	(*TERMINAL 50KF1 (EL6001 Interface (RS232))  ********1-Channel Serial Interface RS232***********************)
	ib50A1_EL6001PortNo								AT %I* :  UINT;
	ist50A1_HandScannerCOMPortDataIn				AT %I* :  EL6InData22B;
	qst50A1_HandScannerCOMPortDataOut				AT %Q*: EL6OutData22B;

	(*TERMINAL 60KF1 (EL1008 8Ch. Dig. Input 24V, 3ms) ******************************************************)
	ib60KF1_1_Spare 								AT %I*: BOOL;
	ib60KF1_5_Spare									AT %I*: BOOL;
	ib60KF1_2_Spare									AT %I*: BOOL;
	ib60KF1_6_Spare									AT %I*: BOOL;
	ib60KF1_3_Spare 								AT %I*: BOOL;
	ib60KF1_7_Spare									AT %I*: BOOL;
	ib60KF1_4_Spare									AT %I*: BOOL;
	ib60KF1_8_Spare 	 							AT %I*: BOOL;

	(*TERMINAL 61KF1 (EL1008 8Ch. Dig. Input 24V, 3ms) ******************************************************)
	ib61KF1_1_DoorOpenZone1_SFCP					AT %I*: BOOL;
	ib61KF1_5_DoorOpenZone2_SFCP					AT %I*: BOOL;
	ib61KF1_2_CasePackerAutoRun_SFCP  				AT %I*: BOOL;
	ib61KF1_6_CaseRejected_SFCP		 				AT %I*: BOOL;
	ib61KF1_3_RowComplete_SFCP  					AT %I*: BOOL;
	ib61KF1_7_LayerComplete_SFCP  					AT %I*: BOOL;
	ib61KF1_4_CaseComplete_SFCP  					AT %I*: BOOL;
	ib61KF1_8_CaseDischarged_SFCP  					AT %I*: BOOL;

	(*TERMINAL 62KF1 (EL1008 8Ch. Dig. Input 24V, 3ms) ******************************************************)
	ib62KF1_1_CasePresentPosition01_SFCP								AT %I*: BOOL;
	ib62KF1_5_CasePresentPosition02_SFCP								AT %I*: BOOL;
	ib62KF1_2_CasePresentPosition03_SFCP						AT %I*: BOOL;
	ib62KF1_6_CasePresentPosition04_SFCP							AT %I*: BOOL;
	ib62KF1_3_CasePresentPosition05_SFCP							AT %I*: BOOL;
	ib62KF1_7_CasePresentPosition06_SFCP							AT %I*: BOOL;
	ib62KF1_4_CasePresentPosition07_SFCP								AT %I*: BOOL;
	ib62KF1_8_CasePresentPosition08_SFCP							AT %I*: BOOL;

	(*TERMINAL 63KF1 (EL1008 8Ch. Dig. Input 24V, 3ms) ******************************************************)
	ib63KF1_1_24VPowerSupplyOK 						AT %I*: BOOL;
	ib63KF1_5_EthernetSwitchOK 						AT %I*: BOOL;	 (* Option *)
	ib63KF1_2_CaseLabelValidationTrig_SFCP 			AT %I*: BOOL;
	ib63KF1_6_QAButtonRejectOuter_SFCP 				AT %I*: BOOL;
	ib63KF1_3_IntermediatePush_SFCP 				AT %I*: BOOL;
	ib63KF1_7_24VPowerSupplyAdditionalUnitOK			AT %I*: BOOL;
	ib63KF1_4_CasePresentPrintAreaSensor			AT %I*: BOOL;	 (* Option *)
	ib63KF1_8_CaseLeavingPrintAreaSensor			AT %I*: BOOL;	 (* Option *)

	(*TERMINAL 64KF1 (EL1008 8Ch. Dig. Input 24V, 3ms) ******************************************************)
	ib64KF1_1_PackSeparationDriveOK					AT %I*: BOOL;
	ib64KF1_5_Spare							AT %I*: BOOL;	(*  *)
	ib64KF1_2_IntermediateCameraTrigSesnorOK						AT %I*: BOOL;	(*  *)
	ib64KF1_6_AdditionalConveyorPlugConnected					AT %I*: BOOL;	(*  *)
	ib64KF1_3_OutfeedConveyorPlugConnected			AT %I*: BOOL; (**)
	ib64KF1_7_TransferConveyorPlugConnected			AT %I*: BOOL;	(* *)
	ib64KF1_4_Guard1 								AT %I*: BOOL; 	(* *)
	ib64KF1_8_Guard2								AT %I*: BOOL; 	(**)

	(*TERMINAL 65KF1 (EL1008 8Ch. Dig. Input 24V, 3ms) ******************************************************)
	ib65KF1_1_PSRisReset							AT %I*: BOOL;
	ib65KF1_5_PSRisOK								AT %I*: BOOL;
	ib65KF1_2_EmergencyStopFromPSR					AT %I*: BOOL;
	ib65KF1_6_EmergencyCircuitFromPSR 				AT %I*: BOOL;
	ib65KF1_3_AirDumpStatus					AT %I*: BOOL; 	(*  *)
	ib65KF1_7_Guard3								AT %I*: BOOL; 	(*  *)
	ib65KF1_4_Guard4								AT %I*: BOOL; 	(*   *)
	ib65KF1_8_Guard5								AT %I*: BOOL; 	(*  *)

	(*TERMINAL 66KF1 (EL1008 8Ch. Dig. Input 24V, 3ms) ******************************************************)
	ib66KF1_1_AirSupplyOK									AT %I*: BOOL;
	ib66KF1_5_PreMachineInAutorun					AT %I*: BOOL;		(*coneccted - input in PreMachine plug 18DX1 *)
	ib66KF1_2_PostMachineInAutorun					AT %I*: BOOL;		(*not coneccted - input in Safety plug 18DX2 *)
	ib66KF1_6_OuterRejectConfirmation				AT %I*: BOOL;		(*Duplicated*)
	ib66KF1_3_MainConveyorStart						AT %I*: BOOL;
	ib66KF1_7_CaseRejctConfirmCameraInReadCycle	AT %I*: BOOL;
	ib66KF1_4_CaseRejctConfirmCameraNoRead		AT %I*: BOOL;
	ib66KF1_8_CaseRejctConfirmCameraGoodRead		AT %I*: BOOL;

	(*TERMINAL 67KF1 (EL1008 8Ch. Dig. Input 24V, 3ms) ******************************************************)
	ib67KF1_1_Spare									AT %I*: BOOL;
	ib67KF1_5_Spare									AT %I*: BOOL;
	ib67KF1_2_Spare									AT %I*: BOOL;
	ib67KF1_6_Spare									AT %I*: BOOL;
	ib67KF1_3_Spare									AT %I*: BOOL;
	ib67KF1_7_Spare									AT %I*: BOOL;
	ib67KF1_4_Spare									AT %I*: BOOL;
	ib67KF1_8_Spare									AT %I*: BOOL;

	(*TERMINAL 69KF1 (EL1008 8Ch. Dig. Input 24V, 3ms) ******************************************************)
	ib69KF1_1_Labeller01Ready							AT %I*: BOOL;
	ib69KF1_5_Labeller01DataReady						AT %I*: BOOL;
	ib69KF1_2_Labeller01HomePosition							AT %I*: BOOL;
	ib69KF1_6_Labeller01LabelPrinted							AT %I*: BOOL;
	ib69KF1_3_Labeller01SummaryWarning							AT %I*: BOOL;
	ib69KF1_7_Labeller01Error								AT %I*: BOOL;
	ib69KF1_4_Labeller01AirPressureOK							AT %I*: BOOL;
	ib69KF1_8_Labeller01InPosition						AT %I*: BOOL;

	(*TERMINAL 70KF1 (EL1008 8Ch. Dig. Input 24V, 3ms) ******************************************************)
	ib70KF1_1_MainsSupplyHealthy					AT %I*: BOOL;	(*  *)
	ib70KF1_5_UPSHealthy							AT %I*: BOOL;	(*  *)
	ib70KF1_2_UPSBatteryMode						AT %I*: BOOL;	(*  *)
	ib70KF1_6_UPSBatteryCharging					AT %I*: BOOL;	(*  *)
	ib70KF1_3_Spare									AT %I*: BOOL; (**)
	ib70KF1_7_Spare								AT %I*: BOOL;	(* *)
	ib70KF1_4_Spare 								AT %I*: BOOL; 	(* *)
	ib70KF1_8_Spare								AT %I*: BOOL; 	(* *)

	(*TERMINAL 80KF1 (EL2008 8Ch. Dig. Output 24V, 0.5A) ******************************************************)
	qb80KF1_1_LightPoleGREEN  						AT %Q*: BOOL;
	qb80KF1_5_LightPoleAMBER  						AT %Q*: BOOL;
	qb80KF1_2_LightPoleRED  						AT %Q*: BOOL;
	qb80KF1_6_LightPoleALARM  						AT %Q*: BOOL;	 (* Option *)
	qb80KF1_3_LightHandscannerBoxGreen 				AT %Q*: BOOL;	 (* Option *)
	qb80KF1_7_LightHandscannerBoxRed  				AT %Q*: BOOL;	 (* Option *)
	qb80KF1_4_Spare  								AT %Q*: BOOL;
	qb80KF1_8_OuterRejectSignal   					AT %Q*: BOOL;	 (*Option*)

	(*TERMINAL 81KF1 (EL2008 8Ch. Dig. Output 24V, 0.5A) ******************************************************)
	qb81KF1_1_SafetyReset	  						AT %Q*: BOOL;
	qb81KF1_5_PackSeperationDriveFaultAck			AT %Q*: BOOL;
	qb81KF1_2_PackSeperationDriveBrakeRelease		AT %Q*: BOOL;	 (* Option *)
	qb81KF1_6_CaseRejctConfirmCameraPower 								AT %Q*: BOOL;
	qb81KF1_3_CaseRejctConfirmCameraTrigger									AT %Q*: BOOL;
	qb81KF1_7_PreMachineAddditionalCutOut			AT %Q*: BOOL;	 (* not coneccted - output in Safety plug 18DX1  *)
	qb81KF1_4_PreMachineCutOut						AT %Q*: BOOL;	(*coneccted - output in PreMachine plug 18DX1 *)
	qb81KF1_8_PostMachineAddditionalCutOut	 					AT %Q*: BOOL;		(* not coneccted - output in PostMachine Safety plug 18DX2 *)

	(*TERMINAL 82KF1 (EL2008 8Ch. Dig. Output 24V, 0.5A) ******************************************************)
	qb82KF1_1_PostMachineCutOut_STCP		  					AT %Q*: BOOL;		(*coneccted - output in PostMachine plug 19DX2 *)
	qb82KF1_5_CaseValidationOK_STCP					AT %Q*: BOOL;
	qb82KF1_2_OuterValidationOK_STCP 				AT %Q*: BOOL;
	qb82KF1_6_CaseContentOK_STCP					AT %Q*: BOOL;
	qb82KF1_3_LabellerInhibit_STL					AT %Q*: BOOL;
	qb82KF1_7_RejectSignal3_STL 					AT %Q*: BOOL;	(*  *)
	qb82KF1_4_Miscellaneous_STL						AT %Q*: BOOL;	(*  *)
	qb82KF1_8_Spare			 						AT %Q*: BOOL;

	(*TERMINAL 83KF1 (EL2008 8Ch. Dig. Output 24V, 0.5A) ******************************************************)
	qb83KF1_1_PackSepparationDriveRun									AT %Q*: BOOL;
	qb83KF1_5_AdditionalConveyor01Run									AT %Q*: BOOL;
	qb83KF1_2_AdditionalConveyor02Run									AT %Q*: BOOL;
	qb83KF1_6_Spare									AT %Q*: BOOL;
	qb83KF1_3_Spare									AT %Q*: BOOL;
	qb83KF1_7_Spare									AT %Q*: BOOL;
	qb83KF1_4_Spare									AT %Q*: BOOL;
	qb83KF1_8_Labeller01DoorGuardOpen			AT %Q*: BOOL;

	(*TERMINAL 84KF1 (EL2008 8Ch. Dig. Output 24V, 0.5A) ******************************************************)
	qb84KF1_1_Spare								AT %Q*: BOOL;
	qb84KF1_5_Spare									AT %Q*: BOOL;
	qb84KF1_2_Spare									AT %Q*: BOOL;
	qb84KF1_6_Spare									AT %Q*: BOOL;
	qb84KF1_3_Spare									AT %Q*: BOOL;
	qb84KF1_7_Spare									AT %Q*: BOOL;
	qb84KF1_4_Spare									AT %Q*: BOOL;
	qb84KF1_8_Spare									AT %Q*: BOOL;

	(*TERMINAL 88KF1 (EL4002 2Ch. Analog Output, 0…10 V, 12 bit) ******************************************************)
	qn88KF1_1_PackSeparationDriveCh1							AT %Q* : INT;
	qn88KF1_2_Spare											AT %Q* : INT;

	(*TERMINAL 90KF1 (EL2624 4Ch. Relay Output, 125 V AC, 30 V DC, 0.5 A AC, 2 A DC)******************)
	qb90KF1_1_Labeller01ResetSignal					AT %Q*: BOOL;		(**)
	qb90KF1_2_Labeller01PrintSignal							AT %Q*: BOOL;		(**)
	qb90KF1_3_Labeller01ApplySignal1						AT %Q*: BOOL;		(**)
	qb90KF1_4_Labeller01ApplySignal2										AT %Q*: BOOL;

	(*TERMINAL 97KF1 - EL6631 -  PROFINET IO Controller ********************************************************)
	ist97KF1_Master01PNetState 						AT %I* : ST_CX_EtherCATMasterPNetState;

	(*DRIVE  3T1  - G120C ************************************************************************************)
	ist3T1_outerseparation							AT %I* : ST_DRIVE_INPUT;
	qst3T1_outerseparation							AT %Q* : ST_DRIVE_OUTPUT;

	(*DRIVE  4T1  - G120C ************************************************************************************)
	ist4T1_transferconveyor							AT %I* : ST_DRIVE_INPUT;
	qst4T1_transferconveyor							AT %Q* : ST_DRIVE_OUTPUT;

	(*DRIVE  5T1  - G120C ************************************************************************************)
	ist5T1_outfeedconveyor							AT %I* : ST_DRIVE_INPUT;
	qst5T1_outfeedconveyor							AT %Q* : ST_DRIVE_OUTPUT;

	(*DRIVE  6T1  - G120C ************************************************************************************)
	ist6T1_additionalconveyor						AT %I* : ST_DRIVE_INPUT;
	qst6T1_additionalconveyor					AT %Q* : ST_DRIVE_OUTPUT;
END_VAR

// ---- Global Variables/InputsOutputs_OC/IOVariablesEUCA_OC.TcGVL
{attribute 'Tc2GvlVarNames'}
VAR_GLOBAL

(*TERMINAL XXXKF1 - EK1100 **********************************************************)

(*TERMINAL 350KF1 (EL6001 Interface (RS232))  ********1-Channel Serial Interface RS232***********************)
	ib350A1_EL6001PortNo								AT %I* :  UINT;
	ist350A1_HandScannerCOMPortDataIn					AT %I* :  EL6InData22B;
	qst350A1_HandScannerCOMPortDataOut					AT %Q*: EL6OutData22B;

(*TERMINAL 351KF1 - EL4002 ******************************************************)
	qn351KF1_1_OuterValidationLightingIntensity			AT %Q* : INT;
	qn351KF1_2_OuterAggregationLightingIntensity		AT %Q* : INT;

(*TERMINAL 352KF1 - EL4002 ******************************************************)
	qn352KF1_1_CaseContentValidationLightingIntensity	AT %Q* : INT;
	qn352KF1_2_LightingIntensity							AT %Q* : INT;

(*TERMINAL 360KF1 - EL1008 ***********************************************************)
	ib360KF1_1_OuterAtInfeed							AT %I* : BOOL;	(* Option *)
	ib360KF1_5_OuterInfeedBlocked						AT %I* : BOOL;	(* Option clamp*)
	ib360KF1_2_OuterAtLabeller							AT %I* : BOOL;	(* Option gate*)
	ib360KF1_6_PackConfirmationCameraTrigSensor			AT %I* : BOOL;
	ib360KF1_3_OuterValidationCameraTrigSensor 					AT %I* : BOOL;
	ib360KF1_7_OuterAtReject							AT %I* : BOOL;
	ib360KF1_4_RejectConfirmation						AT %I* : BOOL;
	ib360KF1_8_RejectBinFull								AT %I* : BOOL;

(*TERMINAL 361KF1 - EL1008 ***********************************************************)
	ib361KF1_1_OuterClampExtended							AT %I* : BOOL;
	ib361KF1_5_OuterGateExtended					AT %I* : BOOL;
	ib361KF1_2_OuterGateRetracted						AT %I* : BOOL;
	ib361KF1_6_OuterGateImpactSensor						AT %I* : BOOL;
	ib361KF1_3_RejectCylinderExtended					AT %I* : BOOL;
	ib361KF1_7_RejectCylinderRetracted					AT %I* : BOOL;
	ib361KF1_4_EUCAExitBlocked										AT %I* : BOOL;	(* Option *)
	ib361KF1_8_EUCABuildBack									AT %I* : BOOL;

(*TERMINAL 362KF1 - EL1008 ************************************************************)
	ib362KF1_1_Labeller02Ready							AT %I*: BOOL;
	ib362KF1_5_Labeller02DataReady						AT %I*: BOOL;
	ib362KF1_2_Labeller02HomePosition 			AT %I*: BOOL;
	ib362KF1_6_Labeller02LabelPrinted						AT %I*: BOOL;
	ib362KF1_3_Labeller02SummaryWarning					AT %I*: BOOL;
	ib362KF1_7_Labeller02Error							AT %I*: BOOL;
	ib362KF1_4_Labeller02AirPressureOK							AT %I*: BOOL;
	ib362KF1_8_Labeller02InPosition					AT %I*: BOOL;	(* ??? *)

(*TERMINAL 363KF1 (EL1008 8Ch. Dig. Input 24V, 3ms) ***************************************)
	ib363KF1_1_QAButtonRejectOuter						AT %I*: BOOL;	(* Option *)
	ib363KF1_5_IntermediatePushSensor					AT %I*: BOOL;
	ib363KF1_2_CaseLabelValidationCameraTrigSensor 		AT %I*: BOOL;
	ib363KF1_6_OuterAggregationCameraTrigSensor			AT %I*: BOOL;	(* *)
	ib363KF1_3_RowCompleteSensor						AT %I*: BOOL;
	ib363KF1_7_LayerCompleteSensor						AT %I*: BOOL;
	ib363KF1_4_CaseCompleteSensor						AT %I*: BOOL;
	ib363KF1_8_CaseDischargedSensor						AT %I*: BOOL;

(*TERMINAL 366KF1 (EL1008 8Ch. Dig. Input 24V, 3ms) ****************************************)
	ib366KF1_1_OuterAtAdditionalConveyor02									AT %I*: BOOL;
	ib366KF1_5_ExitBlockedAdditionalConveyor02									AT %I*: BOOL;
	ib366KF1_2_Spare									AT %I*: BOOL;
	ib366KF1_6_Spare									AT %I*: BOOL;
	ib366KF1_3_Spare									AT %I*: BOOL;
	ib366KF1_7_Spare									AT %I*: BOOL;
	ib366KF1_4_Spare								AT %I*: BOOL;
	ib366KF1_8_RemoteAirSupplyOK									AT %I*: BOOL;

(*TERMINAL 380KF1 - EL2008 (EL2008 8Ch. Dig. Output 24V, 0.5A) ********************************)
	qb380KF1_1_ClampCylinderExtend				AT %Q*: BOOL;
	qb380KF1_5_Spare						 			AT %Q*: BOOL;
	qb380KF1_2_GateCylinderExtend 						AT %Q*: BOOL;		(**)
	qb380KF1_6_GateCylinderRetract	 					AT %Q*: BOOL;		(**)
	qb380KF1_3_RejectCylinderExtend						AT %Q*: BOOL;
	qb380KF1_7_RejectCylinderRetract			  		AT %Q*: BOOL;
	qb380KF1_4_Spare								AT %Q*: BOOL;
	qb380KF1_8_PLCControlledAggCameraLightning			AT %Q*: BOOL; (**)

(*TERMINAL 381KF1 (EL2008 8Ch. Dig. Output 24V, 0.5A) ***************************************)
	qb381KF1_1_RearConfirmationCameraTrigger			AT %Q*: BOOL;
	qb381KF1_5_RearConfirmationCameraPower				AT %Q*: BOOL;
	qb381KF1_2_FrontConfirmationCameraTrigger			AT %Q*: BOOL;
	qb381KF1_6_FrontConfirmationCameraPower	 			AT %Q*: BOOL;
	qb381KF1_3_OuterValidationCameraTrig 					AT %Q*: BOOL;
	qb381KF1_7_OuterValidationCameraPower				AT %Q*: BOOL;
	qb381KF1_4_OuterAggregationCameraTrig					AT %Q*: BOOL;
	qb381KF1_8_OuterAggregationCameraPower					AT %Q*: BOOL;

(*TERMINAL 382KF1 (EL2008 8Ch. Dig. Output 24V, 0.5A) ****************************************)
	qb382KF1_1_CaseContentValidationCameraTrig				AT %Q*: BOOL;
	qb382KF1_5_CaseContentValidationCameraPower			AT %Q*: BOOL;
	qb382KF1_2_CaseLabelValidationCameraTrig				AT %Q*: BOOL;
	qb382KF1_6_CaseLabelValidationCameraPower	 			AT %Q*: BOOL;
	qb382KF1_3_OuterValidationCameraLightning					AT %Q*: BOOL;		(**)
	qb382KF1_7_OuterAggregationCameraLightning				AT %Q*: BOOL;		(**)
	qb382KF1_4_CaseContentValidationCameraLightning			AT %Q*: BOOL;		(**)
	qb382KF1_8_Labeller02DoorGuardOpen				AT %Q*: BOOL;		(**)

(*TERMINAL 390KF1 (EL2624 4Ch. Relay Output, 125 V AC, 30 V DC, 0.5 A AC, 2 A DC)******************)
	qb390KF1_1_Labeller02ResetSignal						AT %Q*: BOOL;
	qb390KF1_2_Labeller02PrintSignal						AT %Q*: BOOL;
	qb390KF1_3_Labeller02ApplySignal1						AT %Q*: BOOL;
	qb390KF1_4_Labeller02ApplySignal2								AT %Q*: BOOL;

END_VAR

// ---- Global Variables/InputsOutputs_OC/IOVariablesPAOL_OC.TcGVL
{attribute 'Tc2GvlVarNames'}
VAR_GLOBAL

(*TERMINAL XXXKF1 - EK1100 ******************************************************)

(*TERMINAL 647KF1 - EL4002 ******************************************************)
	qn647KF1_1_LightingIntensity							AT %Q* : INT;
	qn647KF1_2_Spare									AT %Q* : INT;

(*TERMINAL 660KF1 - EL1008 ******************************************************)
	ib660KF1_1_PackAggregationCameraRigTrigger			AT %I* : BOOL;
	ib660KF1_5_PackAggregationCamera1Trigger				AT %I* : BOOL;
	ib660KF1_2_PackAggregationCamera2Trigger				AT %I* : BOOL;
	ib660KF1_6_PackAggregationCamera3Trigger				AT %I* : BOOL;
	ib660KF1_3_PreMachineBuildBack						AT %I* : BOOL;
	ib660KF1_7_TPDExitBlock								AT %I* : BOOL;
	ib660KF1_4_PackAggregationCamera4Trigger				AT %I* : BOOL;	(* Option *)
	ib660KF1_8_PackIsolatorDrive							AT %I* : BOOL;

(*TERMINAL 680KF1 - EL2008 ******************************************************)
	qb680KF1_1_PackAggregationCamera1Enable				AT %Q* : BOOL;
	qb680KF1_5_PackAggregationCamera2Enable				AT %Q* : BOOL;
	qb680KF1_2_PackAggregationCamera3Enable				AT %Q* : BOOL;
	qb680KF1_6_PackAggregationCamera1Power				AT %Q* : BOOL;
	qb680KF1_3_PackAggregationCamera2Power				AT %Q* : BOOL;
	qb680KF1_7_PackAggregationCamera3Power				AT %Q* : BOOL;
	qb680KF1_4_PackAggregationCamera4Enable				AT %Q* : BOOL;
	qb680KF1_8_PackCamerasLenseAir						AT %Q* : BOOL;

END_VAR

// ---- Global Variables/InputsOutputs_OC/IOVariablesPLAS_OC.TcGVL
{attribute 'Tc2GvlVarNames'}
VAR_GLOBAL

(*TERMINAL XXXKF1 - EK1100 ******************************************************)


(*TERMINAL 747KF1 - EL4002 ******************************************************)
	qn747KF1_1_LightingIntensityPackAggregationCamera							AT %Q* : INT;
	qn747KF1_2_LightingIntensityPackConfirmationCamera							AT %Q* : INT;

(*TERMINAL 748KF1 - EL4002 ******************************************************)
	qn748KF1_1_LightingIntensityMasterListCamera		AT %Q* : INT;
	qn748KF1_2_Spare										AT %Q* : INT;

(*TERMINAL 763KF1 - EL1008 ******************************************************)
	ib763KF1_1_MasterListCameraTrigSensor					AT %I* : BOOL;
	ib763KF1_5_SpareMasterListCameraTrigSensor			AT %I* : BOOL;		(* Option *)
	ib763KF1_2_AggregationCameraTrigSensor				AT %I* : BOOL;
	ib763KF1_6_SpareAggregationCamera1TrigSensor		AT %I* : BOOL;		(* Option *)
	ib763KF1_3_SpareAggregationCamera2TrigSensor		AT %I* : BOOL;		(* Option *)
	ib763KF1_7_PackQueueIndex								AT %I* : BOOL; 		(* Option *)
	ib763KF1_4_StackQueueIndex								AT %I* : BOOL; 		(* Option *)
	ib763KF1_8_SpareIndex											AT %I* : BOOL;

(*TERMINAL 764KF1 - EL1008 ******************************************************)
	ib764KF1_1_OuterIndexComplete							AT %I* : BOOL;
	ib764KF1_5_SpareCameraTrigSesnor						AT %I* : BOOL;		(* Option *)
	ib764KF1_2_Guard1 										AT %I* : BOOL;		(*FOCKE/GD Master list guard*)
	ib764KF1_6_Guard2										AT %I* : BOOL;		(*FOCKE/GD Master list guard*)
	ib764KF1_3_Guard3 										AT %I* : BOOL;		(*FOCKE/GD Aggregation guard*)
	ib764KF1_7_Guard4 										AT %I* : BOOL;		(*FOCKE/GD Aggregationt guard*)
	ib764KF1_4_OuterBrushOpen								AT %I* : BOOL;
	ib764KF1_8_RejectTowerActive							AT %I* : BOOL;

(*TERMINAL 765KF1 (EL1008 8Ch. Dig. Input 24V, 3ms) ******************************************************)
	ib765KF1_1_FilmInPosition 								AT %I*: BOOL;
	ib765KF1_5_SparePrinterTrigger							AT %I*: BOOL;
	ib765KF1_2_IntermediateCamera1TrigSesnor				AT %I*: BOOL;
	ib765KF1_6_HeatTunelPackReject							AT %I*: BOOL;
	ib765KF1_3_OuterAtAdditionalConveyor01 				AT %I*: BOOL;
	ib765KF1_7_IntermediateCamera2TrigSesnor				AT %I*: BOOL;
	ib765KF1_4_OuterAtReject									AT %I*: BOOL;		(*AdditionalConveyor01*)
	ib765KF1_8_RejectConfirmation	 						AT %I*: BOOL;		(*AdditionalConveyor01*)

(*TERMINAL 766KF1 - EL1008 ******************************************************)
	ib766KF1_1_RejectCylinderExtended						AT %I* : BOOL;
	ib766KF1_5_RejectCylinderRetracted						AT %I* : BOOL;		(*  *)
	ib766KF1_2_RejectBinFull 									AT %I* : BOOL;		(*AdditionalConveyor01*)
	ib766KF1_6_ExitBlockedAdditionalConveyor01				AT %I* : BOOL;
	ib766KF1_3_IntermediateCamera3TrigSesnor				AT %I* : BOOL;
	ib766KF1_7_Spare											AT %I* : BOOL;	(*Potentially for GD Additional Master list guard*)
	ib766KF1_4_Spare											AT %I* : BOOL;		(* Guard5 Potentially for GD Wrapper door*)
	ib766KF1_8_Spare											AT %I* : BOOL;			(* Guard6 Potentially for GD Wrapper door*)

(*TERMINAL 767KF1 - EL1008 ******************************************************)
	ib767KF1_1_ConveyorInterfaceInputSignal1				AT %I* : BOOL;
	ib767KF1_5_ConveyorInterfaceInputSignal2				AT %I* : BOOL;		(*  *)
	ib767KF1_2_RejectTower2Active							AT %I* : BOOL;		(**)
	ib767KF1_6_Spare											AT %I* : BOOL;
	ib767KF1_3_Spare											AT %I* : BOOL;
	ib767KF1_7_Spare 											AT %I* : BOOL;
	ib767KF1_4_Spare											AT %I* : BOOL;
	ib767KF1_8_Spare											AT %I* : BOOL;


(*TERMINAL 783KF1 - EL2008 ******************************************************)
	qb783KF1_1_MasterListCameraPower						AT %Q* : BOOL;
	qb783KF1_5_SpareMasterListCameraPower					AT %Q* : BOOL;	(* Option *)
	qb783KF1_2_SpareAggregationCameraPower				AT %Q* : BOOL;	(* Option *)
	qb783KF1_6_AggregationCamera1Power					AT %Q* : BOOL;
	qb783KF1_3_AggregationCamera2Power					AT %Q* : BOOL;
	qb783KF1_7_ConfirmationCamera1Power					AT %Q* : BOOL; 	(* Option *)
	qb783KF1_4_ConfirmationCamera2Power					AT %Q* : BOOL; 	(* Option *)
	qb783KF1_8_PLCControlledAggCamerasLightning			AT %Q* : BOOL;

(*TERMINAL 784KF1 - EL2008 ******************************************************)
	qb784KF1_1_MasterListCameraTrigger						AT %Q* : BOOL;
	qb784KF1_5_SpareMasterListCameraTrigger				AT %Q* : BOOL;	(* Option *)
	qb784KF1_2_AggregationCameraTrigger					AT %Q* : BOOL;
	qb784KF1_6_SpareAggregationCamera1Trigger			AT %Q* : BOOL; 	(* Option *)
	qb784KF1_3_SpareAggregationCamera2Trigger			AT %Q* : BOOL; 	(* Option *)
	qb784KF1_7_ConfirmationCamera1Trigger					AT %Q* : BOOL; 	(* Option *)
	qb784KF1_4_ConfirmationCamera2Trigger					AT %Q* : BOOL; 	(* Option *)
	qb784KF1_8_PLCControlledConfCameraLightning			AT %Q* : BOOL;

(*TERMINAL 785KF1 (EL2008 8Ch. Dig. Output 24V, 3ms) ******************************************************)
	qb785KF1_1_IntermediateCamera1Trigger					AT %Q*: BOOL;
	qb785KF1_5_IntermediateCamera1Power					AT %Q*: BOOL;
	qb785KF1_2_IntermediateCamera2Trigger					AT %Q*: BOOL;
	qb785KF1_6_IntermediateCamera3Power					AT %Q*: BOOL;
	qb785KF1_3_RejectCylinderExtended						AT %Q*: BOOL;			(*AdditionalConveyor01*)
	qb785KF1_7_RjectCylinderRetracted						AT %Q*: BOOL;			(*AdditionalConveyor01*)
	qb785KF1_4_IntermediateCamera3Trigger					AT %Q*: BOOL;
	qb785KF1_8_IntermediateCamera3Power					AT %Q*: BOOL;

(*TERMINAL 786KF1 - EL2008 ******************************************************)
	qb786KF1_1_ConveyorInterfaceOutputSignal1				AT %Q* : BOOL;
	qb786KF1_5_ConveyorInterfaceOutputSignal2				AT %Q* : BOOL;	(* Option *)
	qb786KF1_2_Spare											AT %Q* : BOOL;	(* Option *)
	qb786KF1_6_Spare											AT %Q* : BOOL;
	qb786KF1_3_Spare											AT %Q* : BOOL;
	qb786KF1_7_Spare											AT %Q* : BOOL; 	(* Option *)
	qb786KF1_4_Spare											AT %Q* : BOOL; 	(* Option *)
	qb786KF1_8_PLCControlledMLCamerasLightning			AT %Q* : BOOL;

END_VAR

// ---- Global Variables/InputsOutputs_SFLX/IOVariablesCX_SFLX.TcGVL
{attribute 'Tc2GvlVarNames'}
VAR_GLOBAL
(***************************Terminal States Diagnostic*****************************************************)

	istEtherCATMasterState							AT	%I*	: ST_CX_EtherCATMasterState;
	iaEtherCATSlaveState							AT 	%I*	: ARRAY [0..cMAX_ETHERCAT_SLAVES] OF UINT;

(*****************************Input/Output Cards*********************************************************)

	(*TERMINAL 45KF2 (EK1200-5000 EtherCAT Power supply (2A E-Bus)) ***************************************)

	(*TERMINAL 50KF1 (EL6001 Interface (RS232))  ********1-Channel Serial Interface RS232***********************)
	ib50A1_EL6001PortNo								AT %I* :  UINT;
	ist50A1_HandScannerCOMPortDataIn				AT %I* :  EL6InData22B;
	qst50A1_HandScannerCOMPortDataOut				AT %Q*: EL6OutData22B;

	(*TERMINAL 60KF1 (EL1008 8Ch. Dig. Input 24V, 3ms) ******************************************************)
	ib60KF1_1_Spare 								AT %I*: BOOL;
	ib60KF1_5_Spare									AT %I*: BOOL;
	ib60KF1_2_Spare									AT %I*: BOOL;
	ib60KF1_6_Spare									AT %I*: BOOL;
	ib60KF1_3_Spare 								AT %I*: BOOL;
	ib60KF1_7_Spare									AT %I*: BOOL;
	ib60KF1_4_Spare									AT %I*: BOOL;
	ib60KF1_8_Spare 	 							AT %I*: BOOL;

	(*TERMINAL 61KF1 (EL1008 8Ch. Dig. Input 24V, 3ms) ******************************************************)
	ib61KF1_1_DoorOpenZone1_SFCP					AT %I*: BOOL;
	ib61KF1_5_DoorOpenZone2_SFCP					AT %I*: BOOL;
	ib61KF1_2_CasePackerAutoRun_SFCP  				AT %I*: BOOL;
	ib61KF1_6_CaseRejected_SFCP		 				AT %I*: BOOL;
	ib61KF1_3_RowComplete_SFCP  					AT %I*: BOOL;
	ib61KF1_7_LayerComplete_SFCP  					AT %I*: BOOL;
	ib61KF1_4_CaseComplete_SFCP  					AT %I*: BOOL;
	ib61KF1_8_CaseDischarged_SFCP  					AT %I*: BOOL;

	(*TERMINAL 62KF1 (EL1008 8Ch. Dig. Input 24V, 3ms) ******************************************************)
	ib62KF1_1_Spare									AT %I*: BOOL;
	ib62KF1_5_Spare 								AT %I*: BOOL;
	ib62KF1_2_Spare 								AT %I*: BOOL;
	ib62KF1_6_Spare 								AT %I*: BOOL;
	ib62KF1_3_Spare									AT %I*: BOOL;
	ib62KF1_7_Spare 								AT %I*: BOOL;
	ib62KF1_4_Spare 								AT %I*: BOOL;
	ib62KF1_8_Spare 								AT %I*: BOOL;

	(*TERMINAL 63KF1 (EL1008 8Ch. Dig. Input 24V, 3ms) ******************************************************)
	ib63KF1_1_24VPowerSupplyOK 						AT %I*: BOOL;
	ib63KF1_5_EthernetSwitchOK 						AT %I*: BOOL;	 (* Option *)
	ib63KF1_2_CaseLabelValidationTrig_SFCP 			AT %I*: BOOL;
	ib63KF1_6_QAButtonRejectOuter_SFCP 				AT %I*: BOOL;
	ib63KF1_3_IntermediatePush_SFCP 				AT %I*: BOOL;
	ib63KF1_7_Spare									AT %I*: BOOL;
	ib63KF1_4_CasePresentPrintAreaSensor			AT %I*: BOOL;	 (* Option *)
	ib63KF1_8_CaseLeavingPrintAreaSensor			AT %I*: BOOL;	 (* Option *)

	(*TERMINAL 64KF1 (EL1008 8Ch. Dig. Input 24V, 3ms) ******************************************************)
	ib64KF1_1_MainsSupplyHealthy					AT %I*: BOOL;	(* UPS *)
	ib64KF1_5_UPSHealthy							AT %I*: BOOL;	(* UPS *)
	ib64KF1_2_UPSBatteryMode						AT %I*: BOOL;	(* UPS *)
	ib64KF1_6_UPSBatteryCharging					AT %I*: BOOL;	(* UPS *)
	ib64KF1_3_TransferConveyorPlugConnected			AT %I*: BOOL; (*LARS and SFLX*)
	ib64KF1_7_OutfeedConveyorPlugConnected			AT %I*: BOOL;	(* SFLX*)
	ib64KF1_4_Guard1 								AT %I*: BOOL; 	(* LARS Transfer Coveyor printer*)
	ib64KF1_8_Guard2								AT %I*: BOOL; 	(* LARS Transfer Coveyor or pinch guard*)

	(*TERMINAL 65KF1 (EL1008 8Ch. Dig. Input 24V, 3ms) ******************************************************)
	ib65KF1_1_PSRisReset							AT %I*: BOOL;
	ib65KF1_5_PSRisOK								AT %I*: BOOL;
	ib65KF1_2_EmergencyStopFromPSR					AT %I*: BOOL;
	ib65KF1_6_EmergencyCircuitFromPSR 				AT %I*: BOOL;
	ib65KF1_3_Guard6									AT %I*: BOOL; 	(*  SFLX*)
	ib65KF1_7_Guard3								AT %I*: BOOL; 	(*  SFLX*)
	ib65KF1_4_Guard4								AT %I*: BOOL; 	(*  SFLX *)
	ib65KF1_8_Guard5								AT %I*: BOOL; 	(*  SFLX*)

	(*TERMINAL 66KF1 (EL1008 8Ch. Dig. Input 24V, 3ms) ******************************************************)
	ib66KF1_1_Spare									AT %I*: BOOL;
	ib66KF1_5_PreMachineInAutorun					AT %I*: BOOL;		(*coneccted - input in PreMachine plug 18DX1 *)
	ib66KF1_2_PostMachineInAutorun					AT %I*: BOOL;		(*not coneccted - input in Safety plug 18DX2 *)
	ib66KF1_6_Spare									AT %I*: BOOL;
	ib66KF1_3_Spare									AT %I*: BOOL;
	ib66KF1_7_Spare									AT %I*: BOOL;
	ib66KF1_4_Spare									AT %I*: BOOL;
	ib66KF1_8_Spare									AT %I*: BOOL;

	(*TERMINAL 67KF1 (EL1008 8Ch. Dig. Input 24V, 3ms) ******************************************************)
	ib67KF1_1_Spare									AT %I*: BOOL;
	ib67KF1_5_Spare									AT %I*: BOOL;
	ib67KF1_2_Spare									AT %I*: BOOL;
	ib67KF1_6_Spare									AT %I*: BOOL;
	ib67KF1_3_Spare									AT %I*: BOOL;
	ib67KF1_7_Spare									AT %I*: BOOL;
	ib67KF1_4_Spare									AT %I*: BOOL;
	ib67KF1_8_Spare									AT %I*: BOOL;

	(*TERMINAL 68KF1 (EL1008 8Ch. Dig. Input 24V, 3ms) ******************************************************)
	ib68KF1_1_ReadyToPrint							AT %I*: BOOL;		(*M-Series Printer Ready*)
	ib68KF1_5_BufferNotEmpty						AT %I*: BOOL;		(*M-Series Data Ready*)
	ib68KF1_2_PrintDone								AT %I*: BOOL;		(*M-Series Label Printed*)
	ib68KF1_6_PrinterWarning							AT %I*: BOOL;		(*M-Series Summary Warningy*)
	ib68KF1_3_PrinterError							AT %I*: BOOL;		(*M-Series Summary Error*)
	ib68KF1_7_Spare									AT %I*: BOOL;
	ib68KF1_4_AdditionalConveyorPlugConnected	AT %I*: BOOL;
	ib68KF1_8_Spare									AT %I*: BOOL;

	(*TERMINAL 80KF1 (EL2008 8Ch. Dig. Output 24V, 0.5A) ******************************************************)
	qb80KF1_1_LightPoleGREEN  						AT %Q*: BOOL;
	qb80KF1_5_LightPoleAMBER  						AT %Q*: BOOL;
	qb80KF1_2_LightPoleRED  						AT %Q*: BOOL;
	qb80KF1_6_LightPoleALARM  						AT %Q*: BOOL;	 (* Option *)
	qb80KF1_3_LightHandscannerBoxGreen 				AT %Q*: BOOL;	 (* Option *)
	qb80KF1_7_LightHandscannerBoxRed  				AT %Q*: BOOL;	 (* Option *)
	qb80KF1_4_Spare  								AT %Q*: BOOL;
	qb80KF1_8_OuterRejectSignal   					AT %Q*: BOOL;	 (*Option nie uzywamy*)

	(*TERMINAL 81KF1 (EL2008 8Ch. Dig. Output 24V, 0.5A) ******************************************************)
	qb81KF1_1_SafetyReset	  						AT %Q*: BOOL;
	qb81KF1_5_Spare 								AT %Q*: BOOL;
	qb81KF1_2_PackSeperationDriveBrakeRelease		AT %Q*: BOOL;	 (* Option *)
	qb81KF1_6_Spare 								AT %Q*: BOOL;
	qb81KF1_3_Spare									AT %Q*: BOOL;
	qb81KF1_7_PreMachineAddditionalCutOut			AT %Q*: BOOL;	 (* Option *)
	qb81KF1_4_PreMachineCutOut						AT %Q*: BOOL;(*coneccted - output in PreMachine plug 18DX1 *)
	qb81KF1_8_PostMachineRun	 					AT %Q*: BOOL;		(* not coneccted - output in Safety plug 18DX2 *)

	(*TERMINAL 82KF1 (EL2008 8Ch. Dig. Output 24V, 0.5A) ******************************************************)
	qb82KF1_1_CutOut_STCP		  					AT %Q*: BOOL;
	qb82KF1_5_CaseValidationOK_STCP					AT %Q*: BOOL;
	qb82KF1_2_OuterValidationOK_STCP 				AT %Q*: BOOL;
	qb82KF1_6_CaseContentOK_STCP					AT %Q*: BOOL;
	qb82KF1_3_LabellerInhibit_STL					AT %Q*: BOOL;
	qb82KF1_7_RejectSignal3_STL 					AT %Q*: BOOL;	(* Option *)
	qb82KF1_4_Miscellaneous_STL						AT %Q*: BOOL;	(* Option *)
	qb82KF1_8_Spare			 						AT %Q*: BOOL;

	(*TERMINAL 83KF1 (EL2008 8Ch. Dig. Output 24V, 0.5A) ******************************************************)
	qb83KF1_1_Spare									AT %Q*: BOOL;
	qb83KF1_5_Spare									AT %Q*: BOOL;
	qb83KF1_2_Spare									AT %Q*: BOOL;
	qb83KF1_6_Spare									AT %Q*: BOOL;
	qb83KF1_3_Spare									AT %Q*: BOOL;
	qb83KF1_7_Spare									AT %Q*: BOOL;
	qb83KF1_4_Spare									AT %Q*: BOOL;
	qb83KF1_8_Spare			 						AT %Q*: BOOL;

	(*TERMINAL 90KF1 (EL2624 4Ch. Relay Output, 125 V AC, 30 V DC, 0.5 A AC, 2 A DC)******************)
	qb90KF1_1_PrintingEnableSignal						AT %Q*: BOOL;		(*M-Series Print*)
	qb90KF1_2_AlarmQuiteSignal							AT %Q*: BOOL;		(*M-Series Reset*)
	qb90KF1_3_ProductDetectSignal						AT %Q*: BOOL;		(*M-Series Apply*)
	qb90KF1_4_Spare										AT %Q*: BOOL;


	(*TERMINAL 97KF1 - EL6631 -  PROFINET IO Controller ********************************************************)
	ist97KF1_Master01PNetState 						AT %I* : ST_CX_EtherCATMasterPNetState;

	(*DRIVE  3T1  - G120C ************************************************************************************)
	ist3T1_outerseparation							AT %I* : ST_DRIVE_INPUT;
	qst3T1_outerseparation							AT %Q* : ST_DRIVE_OUTPUT;

	(*DRIVE  4T1  - G120C ************************************************************************************)
	ist4T1_transferconveyor							AT %I* : ST_DRIVE_INPUT;
	qst4T1_transferconveyor							AT %Q* : ST_DRIVE_OUTPUT;

	(*DRIVE  5T1  - G120C ************************************************************************************)
	ist5T1_outfeedconveyor							AT %I* : ST_DRIVE_INPUT;
	qst5T1_outfeedconveyor							AT %Q* : ST_DRIVE_OUTPUT;

	(*DRIVE  6T1  - G120C ************************************************************************************)
	ist6T1_additionalconveyor						AT %I* : ST_DRIVE_INPUT;
	qst6T1_additionalconveyor					AT %Q* : ST_DRIVE_OUTPUT;
END_VAR

// ---- Global Variables/InputsOutputs_SFLX/IOVariablesEUCA_SFLX.TcGVL
{attribute 'Tc2GvlVarNames'}
VAR_GLOBAL

(*TERMINAL XXXKF1 - EK1100 **********************************************************)

(*ENCODER 333P2 - SICK AFS60A  ******************************************************)
	in333P2_PositionValue						AT %I* : UDINT;
	in333P2_RawPositionValue					AT %I* : UDINT;
	in333P2_AlarmStatus							AT %I* : UINT;
	in333P2_WarningStatus						AT %I* : UINT;

(*TERMINAL 349KF1 - EL4002 ******************************************************)
	qn349KF1_1_LightingIntensityTop						AT %Q* : INT;
	qn349KF1_2_LightingIntensityBottom					AT %Q* : INT;

(*TERMINAL 350KF1 (EL6001 Interface (RS232))  ********1-Channel Serial Interface RS232***********************)
	ib350A1_EL6001PortNo								AT %I* :  UINT;
	ist350A1_HandScannerCOMPortDataIn					AT %I* :  EL6InData22B;
	qst350A1_HandScannerCOMPortDataOut					AT %Q*: EL6OutData22B;

(*TERMINAL 351KF1 - EL4002 ******************************************************)
	qn351KF1_1_OuterValidationLightingIntensity						AT %Q* : INT;
	qn351KF1_2_OuterAggregationLightingIntensity				AT %Q* : INT;

(*TERMINAL 352KF1 - EL4002 ******************************************************)
	qn352KF1_1_CaseContentValidationLightingIntensity		AT %Q* : INT;
	qn352KF1_2_LightingIntensity							AT %Q* : INT;

(*TERMINAL 360KF1 - EL1008 ***********************************************************)
	ib360KF1_1_OuterAtInfeed							AT %I* : BOOL;	(* Option *)
	ib360KF1_5_OuterInfeedBlocked						AT %I* : BOOL;	(* Option *)
	ib360KF1_2_OuterAtLabeller							AT %I* : BOOL;
	ib360KF1_6_PackConfirmationCameraTrigSensor			AT %I* : BOOL;
	ib360KF1_3_OuterMasterListTrigSensor 					AT %I* : BOOL;
	ib360KF1_7_OuterAtReject							AT %I* : BOOL;
	ib360KF1_4_RejectConfirmation						AT %I* : BOOL;
	ib360KF1_8_RejectBinFull								AT %I* : BOOL;

(*TERMINAL 361KF1 - EL1008 ***********************************************************)
	ib361KF1_1_OuterGateExtended							AT %I* : BOOL;
	ib361KF1_5_OuterGateRetracted					AT %I* : BOOL;
	ib361KF1_2_FirstPusherExtended						AT %I* : BOOL;
	ib361KF1_6_FirstPusherRetracted						AT %I* : BOOL;
	ib361KF1_3_RejectCylinderExtended					AT %I* : BOOL;
	ib361KF1_7_RejectCylinderRetracted					AT %I* : BOOL;
	ib361KF1_4_SecondPusherExtended						AT %I* : BOOL;	(* Option *)
	ib361KF1_8_SecondPusherRetracted						AT %I* : BOOL;

(*TERMINAL 362KF1 - EL1008 ************************************************************)
	ib362KF1_1_Labeller01Ready							AT %I*: BOOL;
	ib362KF1_5_Labeller01DataReady						AT %I*: BOOL;
	ib362KF1_2_Labeller01ApplicatorHomePosition 			AT %I*: BOOL;
	ib362KF1_6_Labeller01LabelPrinted						AT %I*: BOOL;
	ib362KF1_3_Labeller01SummaryWarning					AT %I*: BOOL;
	ib362KF1_7_Labeller01Error							AT %I*: BOOL;
	ib362KF1_4_AirPressureOK							AT %I*: BOOL;
	ib362KF1_8_Labeller01InPosition					AT %I*: BOOL;	(* ??? *)

(*TERMINAL 363KF1 (EL1008 8Ch. Dig. Input 24V, 3ms) ***************************************)
	ib363KF1_1_QAButtonRejectOuter						AT %I*: BOOL;	(* Option *)
	ib363KF1_5_IntermediatePushSensor					AT %I*: BOOL;
	ib363KF1_2_CaseLabelValidationCameraTrigSensor	AT %I*: BOOL;
	ib363KF1_6_CaseAtRejectStation						AT %I*: BOOL;	(* Option *)
	ib363KF1_3_RowCompleteSensor						AT %I*: BOOL;
	ib363KF1_7_LayerCompleteSensor						AT %I*: BOOL;
	ib363KF1_4_CaseCompleteSensor						AT %I*: BOOL;
	ib363KF1_8_CaseDischargedSensor						AT %I*: BOOL;

(*TERMINAL 364KF1 (EL1008 8Ch. Dig. Input 24V, 3ms) ****************************************)
	ib364KF1_1_AdditionalRejectCylExtended				AT %I*: BOOL;
	ib364KF1_5_AdditionalRejectCylRetracted				AT %I*: BOOL;
	ib364KF1_2_OuterInfeedJam							AT %I*: BOOL;
	ib364KF1_6_PackAggregationCameraRigTrigger		AT %I*: BOOL;
	ib364KF1_3_OuterAtSideFlexExit						AT %I*: BOOL;
	ib364KF1_7_OuterTransferConfirmation				AT %I*: BOOL;
	ib364KF1_4_EUCAExitBlocked								AT %I*: BOOL;
	ib364KF1_8_EUCABuildBack							AT %I*: BOOL;

(*TERMINAL 365KF1 (EL1008 8Ch. Dig. Input 24V, 3ms) ****************************************)
	ib365KF1_1_OuterAtPostMachineInfeed				AT %I*: BOOL;
	ib365KF1_5_RejectConfirmationNCW				AT %I*: BOOL;
	ib365KF1_2_RejectBinFullNCW						AT %I*: BOOL;
	ib365KF1_6_OuterReadingConfirmation			AT %I*: BOOL;
	ib365KF1_3_OuterAtTransferReject				AT %I*: BOOL;
	ib365KF1_7_Spare									AT %I*: BOOL;
	ib365KF1_4_Spare									AT %I*: BOOL;
	ib365KF1_8_Spare									AT %I*: BOOL;

(*TERMINAL 366KF1 (EL1008 8Ch. Dig. Input 24V, 3ms) ****************************************)
	ib366KF1_1_Spare									AT %I*: BOOL;
	ib366KF1_5_Spare									AT %I*: BOOL;
	ib366KF1_2_Spare									AT %I*: BOOL;
	ib366KF1_6_Spare									AT %I*: BOOL;
	ib366KF1_3_Spare									AT %I*: BOOL;
	ib366KF1_7_Spare									AT %I*: BOOL;
	ib366KF1_4_Spare									AT %I*: BOOL;
	ib366KF1_8_Spare									AT %I*: BOOL;

(*TERMINAL 380KF1 - EL2008 (EL2008 8Ch. Dig. Output 24V, 0.5A) ********************************)
	qb380KF1_1_FirstPusherCylinderExtend				AT %Q*: BOOL;
	qb380KF1_5_SecondPusherCylinderExtend	 			AT %Q*: BOOL;
	qb380KF1_2_GateCylinderExtend 						AT %Q*: BOOL;		(*Additional reject acturator for SFLX*)
	qb380KF1_6_GateCylinderRetract	 					AT %Q*: BOOL;		(*Additional reject acturator for SFLX*)
	qb380KF1_3_RejectCylinderExtend						AT %Q*: BOOL;
	qb380KF1_7_RejectCylinderRetract			  		AT %Q*: BOOL;
	qb380KF1_4_FirstPusherCylinderRetract				AT %Q*: BOOL;
	qb380KF1_8_SecondPusherCylinderRetract				AT %Q*: BOOL;

(*TERMINAL 381KF1 (EL2008 8Ch. Dig. Output 24V, 0.5A) ***************************************)
	qb381KF1_1_RearConfirmationCameraTrigger			AT %Q*: BOOL;
	qb381KF1_5_RearConfirmationCameraPower				AT %Q*: BOOL;
	qb381KF1_2_FrontConfirmationCameraTrigger			AT %Q*: BOOL;
	qb381KF1_6_FrontConfirmationCameraPower	 			AT %Q*: BOOL;
	qb381KF1_3_OuterValidationCameraTrig 					AT %Q*: BOOL;
	qb381KF1_7_OuterValidationCameraPower				AT %Q*: BOOL;
	qb381KF1_4_OuterAggregationCameraTrig					AT %Q*: BOOL;
	qb381KF1_8_OuterAggregationCameraPower					AT %Q*: BOOL;

(*TERMINAL 382KF1 (EL2008 8Ch. Dig. Output 24V, 0.5A) ****************************************)
	qb382KF1_1_CaseContentValidationCameraTrig				AT %Q*: BOOL;
	qb382KF1_5_CaseContentValidationCameraPower			AT %Q*: BOOL;
	qb382KF1_2_CaseLabelValidationCameraTrig				AT %Q*: BOOL;
	qb382KF1_6_CaseLabelValidationCameraPower	 			AT %Q*: BOOL;
	qb382KF1_3_PackAggregationCamera1Trigger			AT %Q*: BOOL;		(*Used for SFLX*)
	qb382KF1_7_PackAggregationCamera1Power				AT %Q*: BOOL;		(*Used for SFLX*)
	qb382KF1_4_PackAggregationCamera2Trigger			AT %Q*: BOOL;		(*Used for SFLX*)
	qb382KF1_8_PackAggregationCamera2Power				AT %Q*: BOOL;		(*Used for SFLX*)

(*TERMINAL 383KF1 (EL2008 8Ch. Dig. Output 24V, 0.5A) ****************************************)
	qb383KF1_1_LightPoleGREEN						AT %Q*: BOOL;
	qb383KF1_5_LightPoleAMBER						AT %Q*: BOOL;
	qb383KF1_2_LightPoleRED						AT %Q*: BOOL;
	qb383KF1_6_LightPoleALARM						AT %Q*: BOOL;
	qb383KF1_3_OuterContentValidationCameraTrig			AT %Q*: BOOL;
	qb383KF1_7_OuterContentValidationCameraPower	AT %Q*: BOOL;
	qb383KF1_4_RejectActiveNCW										AT %Q*: BOOL;
	qb383KF1_8_Spare									AT %Q*: BOOL;

(*TERMINAL 384KF1 (EL2008 8Ch. Dig. Output 24V, 0.5A) ****************************************)
	qb384KF1_1_Spare										AT %Q*: BOOL;
	qb384KF1_5_Spare										AT %Q*: BOOL;
	qb384KF1_2_Spare										AT %Q*: BOOL;
	qb384KF1_6_Spare										AT %Q*: BOOL;
	qb384KF1_3_PLCControlledOuterValidCamLightning		AT %Q*: BOOL;
	qb384KF1_7_PLCControlledOuterAggCamLightning		AT %Q*: BOOL;
	qb384KF1_4_PLCControlledCaseContentCamLightning	AT %Q*: BOOL;
	qb384KF1_8_Spare									AT %Q*: BOOL;

(*TERMINAL 390KF1 (EL2624 4Ch. Relay Output, 125 V AC, 30 V DC, 0.5 A AC, 2 A DC)******************)
	qb390KF1_1_Labeller1ResetSignal						AT %Q*: BOOL;
	qb390KF1_2_Labeller1PrintSignal						AT %Q*: BOOL;
	qb390KF1_3_Labeller1ApplySignal						AT %Q*: BOOL;
	qb390KF1_4_DoorGuardOK								AT %Q*: BOOL;

END_VAR

// ---- Global Variables/InputsOutputs_SFLX/IOVariablesPAOL_SFLX.TcGVL
{attribute 'Tc2GvlVarNames'}
VAR_GLOBAL

(*TERMINAL XXXKF1 - EK1100 ******************************************************)

(*TERMINAL 647KF1 - EL4002 ******************************************************)
	qn647KF1_1_LightingIntensity							AT %Q* : INT;
	qn647KF1_2_Spare									AT %Q* : INT;

(*TERMINAL 660KF1 - EL1008 ******************************************************)
	ib660KF1_1_PackAggregationCameraRigTrigger			AT %I* : BOOL;
	ib660KF1_5_PackAggregationCamera1Trigger				AT %I* : BOOL;
	ib660KF1_2_PackAggregationCamera2Trigger				AT %I* : BOOL;
	ib660KF1_6_PackAggregationCamera3Trigger				AT %I* : BOOL;
	ib660KF1_3_PreMachineBuildBack						AT %I* : BOOL;
	ib660KF1_7_TPDExitBlock								AT %I* : BOOL;
	ib660KF1_4_PackAggregationCamera4Trigger				AT %I* : BOOL;	(* Option *)
	ib660KF1_8_PackIsolatorDrive							AT %I* : BOOL;

(*TERMINAL 680KF1 - EL2008 ******************************************************)
	qb680KF1_1_PackAggregationCamera1Enable				AT %Q* : BOOL;
	qb680KF1_5_PackAggregationCamera2Enable				AT %Q* : BOOL;
	qb680KF1_2_PackAggregationCamera3Enable				AT %Q* : BOOL;
	qb680KF1_6_PackAggregationCamera1Power				AT %Q* : BOOL;
	qb680KF1_3_PackAggregationCamera2Power				AT %Q* : BOOL;
	qb680KF1_7_PackAggregationCamera3Power				AT %Q* : BOOL;
	qb680KF1_4_PackAggregationCamera4Enable				AT %Q* : BOOL;
	qb680KF1_8_PackCamerasLenseAir						AT %Q* : BOOL;

END_VAR

// ---- Global Variables/InputsOutputs_SFLX/IOVariablesPLAS_SFLX.TcGVL
{attribute 'Tc2GvlVarNames'}
VAR_GLOBAL

(*TERMINAL XXXKF1 - EK1100 ******************************************************)

(*TERMINAL 649KF1 - EL4002 ******************************************************)
	qn649KF1_1_PackAggregationLightingIntensity				AT %Q* : INT;
	qn649KF1_2_LightingIntensity								AT %Q* : INT;

(*TERMINAL 663KF1 - EL1008 ******************************************************)
	ib663KF1_1_MasterListCameraTrigSensor					AT %I* : BOOL;
	ib663KF1_5_SpareMasterListCameraTrigSensor			AT %I* : BOOL;		(* Option *)
	ib663KF1_2_AggregationCameraTrigSensor				AT %I* : BOOL;
	ib663KF1_6_SpareAggregationCamera1TrigSensor		AT %I* : BOOL;		(* Option *)
	ib663KF1_3_SpareAggregationCamera2TrigSensor		AT %I* : BOOL;		(* Option *)
	ib663KF1_7_PackQueueIndex								AT %I* : BOOL; 		(* Option *)
	ib663KF1_4_StackQueueIndex								AT %I* : BOOL; 		(* Option *)
	ib663KF1_8_Spare											AT %I* : BOOL;

(*TERMINAL 664KF1 - EL1008 ******************************************************)
	ib664KF1_1_OuterIndexComplete							AT %I* : BOOL;
	ib664KF1_5_IntermediateCameraTrigSensor				AT %I* : BOOL;		(* TO DO Intemediat Camera Trigger *)
	ib664KF1_2_Guard1 										AT %I* : BOOL;
	ib664KF1_6_Guard2										AT %I* : BOOL;
	ib664KF1_3_Guard3 										AT %I* : BOOL;
	ib664KF1_7_Guard4 										AT %I* : BOOL;
	ib664KF1_4_OuterBrushOpen								AT %I* : BOOL;
	ib664KF1_8_RejectTowerActive							AT %I* : BOOL;

(*TERMINAL 665KF1 (EL1008 8Ch. Dig. Input 24V, 3ms) ******************************************************)
	ib665KF1_1_FilmInPosition 								AT %I*: BOOL;
	ib665KF1_5_IntermediatePrinterTrigger					AT %I*: BOOL;
	ib665KF1_2_Spare									AT %I*: BOOL;
	ib665KF1_6_Spare									AT %I*: BOOL;
	ib665KF1_3_Spare 								AT %I*: BOOL;
	ib665KF1_7_Spare									AT %I*: BOOL;
	ib665KF1_4_Spare									AT %I*: BOOL;
	ib665KF1_8_Spare 	 							AT %I*: BOOL;

(*TERMINAL 683KF1 - EL2008 ******************************************************)
	qb683KF1_1_MasterListCameraPower						AT %Q* : BOOL;
	qb683KF1_5_SpareMasterListCameraPower				AT %Q* : BOOL;	(* Option *)
	qb683KF1_2_SpareAggregationCameraPower				AT %Q* : BOOL;	(* Option *)
	qb683KF1_6_AggregationCamera1Power					AT %Q* : BOOL;
	qb683KF1_3_AggregationCamera2Power					AT %Q* : BOOL;
	qb683KF1_7_ConfirmationCamera1Power					AT %Q* : BOOL; 	(* Option *)
	qb683KF1_4_ConfirmationCamera2Power					AT %Q* : BOOL; 	(* Option *)
	qb683KF1_8_PLCControlledPackAggCamLightning		AT %Q* : BOOL;

(*TERMINAL 684KF1 - EL2008 ******************************************************)
	qb684KF1_1_MasterListCameraTrigger					AT %Q* : BOOL;
	qb684KF1_5_SpareMasterListCameraTrigger				AT %Q* : BOOL;	(* Option *)
	qb684KF1_2_AggregationCameraTrigger					AT %Q* : BOOL;
	qb684KF1_6_SpareAggregationCamera1Trigger			AT %Q* : BOOL; 	(* Option *)
	qb684KF1_3_SpareAggregationCamera2Trigger			AT %Q* : BOOL; 	(* Option *)
	qb684KF1_7_ConfirmationCamera1Trigger				AT %Q* : BOOL; 	(* Option *)
	qb684KF1_4_ConfirmationCamera2Trigger				AT %Q* : BOOL; 	(* Option *)
	qb684KF1_8_Spare											AT %Q* : BOOL;

(*TERMINAL 685KF1 (EL2008 8Ch. Dig. Output 24V, 3ms) ******************************************************)
	qb685KF1_1_IntermediateCameraTrigger								AT %Q*: BOOL;
	qb685KF1_5_IntermediateCameraPower									AT %Q*: BOOL;
	qb685KF1_2_Spare									AT %Q*: BOOL;
	qb685KF1_6_Spare									AT %Q*: BOOL;
	qb685KF1_3_Spare								AT %Q*: BOOL;
	qb685KF1_7_Spare								AT %Q*: BOOL;
	qb685KF1_4_Spare										AT %Q*: BOOL;
	qb685KF1_8_Spare 							AT %Q*: BOOL;

END_VAR

// ---- Global Variables/gIOFiltered.TcGVL
{attribute 'qualified_only'}
{attribute 'Tc2GvlVarNames'}
VAR_GLOBAL

(*METS Serial Filtered Inputs ***************************************************************************************************************)

	stEmptyCOMPortDataIn		: EL6InData22B;		(* linked to the EL60xx in the TwinCAT System Manager *)
	stEmptyCOMPortDataOut		: EL6OutData22B;	(* linked to the EL60xx in the TwinCAT System Manager *)

(*DRIVE - G120C ******************************************************)
	stEmpty_DriveInput			: ST_DRIVE_INPUT;
	stEmpty_DriveOutput			: ST_DRIVE_OUTPUT;

(*METS Safety Filtered Inputs ***************************************************************************************************************)

	stMetsStart					: ST_IO2_InputPLC;
	stMetsStop					: ST_IO2_InputPLC;
	stMetsReset					: ST_IO2_InputPLC;

(*METS Safety Filtered Inputs ***************************************************************************************************************)

	stPSR_IsReset				: ST_IO2_InputPLC;
	stPSR_OK					: ST_IO2_InputPLC;
	stEmergencyStop				: ST_IO2_InputPLC;
	stEmergencyCircuit			: ST_IO2_InputPLC;
	stMotorInverterOK			: ST_IO2_InputPLC;
	stGuardDoorOK				: ST_IO2_InputPLC;

(*METS General Filtered Inputs ***************************************************************************************************************)

	stMETS_24VPowerSupplyOK			: ST_IO2_InputPLC;
	stTPD24VPowerSupplyOK			: ST_IO2_InputPLC;
	stAirPressureOK					: ST_IO2_InputPLC;
	stAirConditionerOK				: ST_IO2_InputPLC;
	stUPSBatteryAlarm				: ST_IO2_InputPLC;
	stNetworkOKFromSwitch			: ST_IO2_InputPLC;

	stDoorOpenZone1					: ST_IO2_InputPLC;
	stDoorOpenZone2					: ST_IO2_InputPLC;

	stCaseAtRejectStation	 		: ST_IO2_InputPLC;
	stCaseRejectedByCasePacker		: ST_IO2_InputPLC;
	stCaseContentValidationComplete	: ST_IO2_InputPLC;
	stCaseLeavingPrintArea			: ST_IO2_InputPLC;


(*METS CX UPS  Filtered Inputs ***************************************************************************************************************)

	stMainSupplyHealthy				: ST_IO2_InputPLC;	
	stUPSHealthy					: ST_IO2_InputPLC;
	stUPSBatteryMode				: ST_IO2_InputPLC;
	stUPSBatteryCharging			: ST_IO2_InputPLC;

(*METS Camera Filtered Inputs ***************************************************************************************************************)

	stCamera01				: ST_IO2_InputPLC;
	stCamera02				: ST_IO2_InputPLC;
	stCamera03				: ST_IO2_InputPLC;
	stCamera04				: ST_IO2_InputPLC;
	stCamera05				: ST_IO2_InputPLC;
	stCamera06				: ST_IO2_InputPLC;
	stCamera07				: ST_IO2_InputPLC;
	stCamera08				: ST_IO2_InputPLC;
	stCamera09				: ST_IO2_InputPLC;
	stCamera10				: ST_IO2_InputPLC;
	stCamera11				: ST_IO2_InputPLC;
	stCamera12				: ST_IO2_InputPLC;

(*METS Casepacker  Filtered Inputs ***************************************************************************************************************)

	stPreMachineAutoRun			: ST_IO2_InputPLC;
	stCasePackerAutoRun			: ST_IO2_InputPLC;

	stEUCAExitBlocked			: ST_IO2_InputPLC;
	stEUCABuildBackPreMachine	: ST_IO2_InputPLC;
	stQAButtonReject			: ST_IO2_InputPLC;

	stOuterAtSystemInfeed		: ST_IO2_InputPLC;
	stOuterAtAdditionalConv		: ST_IO2_InputPLC;

	(*Transfer Conveyor*)
	stTransferCoveyorDoorGuard1			: ST_IO2_InputPLC;
	stTransferCoveyorDoorGuard2			: ST_IO2_InputPLC;

	stTransferConveyorPlugConnected		: ST_IO2_InputPLC;
	stOutfeedConveyorPlugConnected		: ST_IO2_InputPLC;
	stAdditionalConveyorPlugConnected	: ST_IO2_InputPLC;

	stOuterAtRejectStation 				: ST_IO2_InputPLC;
	stOuterRejectConfirm				: ST_IO2_InputPLC;
	stRejectBinFull						: ST_IO2_InputPLC;

	stAuxRowCompleteSesnor		: ST_IO2_InputPLC;
	stRowComplete				: ST_IO2_InputPLC;
	stLayerComplete				: ST_IO2_InputPLC;
	stIntermediatePush			: ST_IO2_InputPLC;
	stCaseComplete				: ST_IO2_InputPLC;
	stCaseDischarged			: ST_IO2_InputPLC;
	stCaseLabelValidation		: ST_IO2_InputPLC;

(*METS Cylinders Filtered Inputs  FB***************************************************************************************************************)

	stClampCylinderExtended					: ST_IO2_InputPLC;
	stClampCylinderRetracted				: ST_IO2_InputPLC;

	stGateCylinderExtended					: ST_IO2_InputPLC;
	stGateCylinderRetracted 				: ST_IO2_InputPLC;

	stRejectCylinderExtended				: ST_IO2_InputPLC;
	stRejectCylinderRetracted 				: ST_IO2_InputPLC;

	stAdditionalRejectCylinderExtended		: ST_IO2_InputPLC;
	stAdditionalRejectCylinderRetracted 	: ST_IO2_InputPLC;

	stFirstPusherCylinderExtended			: ST_IO2_InputPLC;
	stFirstPusherCylinderRetracted 			: ST_IO2_InputPLC;

	stSecondPusherCylinderExtended			: ST_IO2_InputPLC;
	stSecondPusherCylinderRetracted 		: ST_IO2_InputPLC;

(*METS SFLX Machine Filtered Inputs ***************************************************************************************************************)

	stOuterInfeedJam						: ST_IO2_InputPLC;
	stOuterTransferConfirmation				: ST_IO2_InputPLC;
	stRejectConfirmationNCW					: ST_IO2_InputPLC;
	stRejectBinFullNCW						: ST_IO2_InputPLC;
	stOuterAtTransferReject					: ST_IO2_InputPLC;
	stOuterAtSideFlexExit					: ST_IO2_InputPLC;
	stOuterAtPostMachineInfeed				: ST_IO2_InputPLC;

	stGuard1FlexInfeedDoor  				: ST_IO2_InputPLC;
	(*stGuard2FlexPrinterInPositon			: ST_IO2_InputPLC;   (*Printer in Position stLabeller1InPosition	 *) *)
	stGuard3FlexRHDoor						: ST_IO2_InputPLC;
	stGuard4FlexPrinterDoor					: ST_IO2_InputPLC;
	stGuard5FlexLHDoor						:	ST_IO2_InputPLC;

(*METS CML Filtered Inputs ***************************************************************************************************************)

	stGuard1UpperSideAccessDoor			: ST_IO2_InputPLC;
	stGuard2UpperDoorLabellerSide		: ST_IO2_InputPLC;
	stGuard3OutfeedTunnel				: ST_IO2_InputPLC;
	stGuard4ElectricalBoxInPosition		: ST_IO2_InputPLC;
	stGuard5RejectBinLHSide				: ST_IO2_InputPLC;
	stGuard6RejectBinRHSide				: ST_IO2_InputPLC;
	stGuard7HTTDoorGuard				: ST_IO2_InputPLC;

	stGuard10FrontUpperDoor				: ST_IO2_InputPLC;
	stGuard11GuardLowerLabellerSide		: ST_IO2_InputPLC;

	stRejectBinGuardIsReset				: ST_IO2_InputPLC;
	stLabeller1GuardIsReset				: ST_IO2_InputPLC;
	stLabeller2GuardIsReset				: ST_IO2_InputPLC;

	stResetPB							: ST_IO2_InputPLC;
	stOuterAtCMLRejectStation			: ST_IO2_InputPLC;

	stRotaryTransferPackAtStopPlate		: ST_IO2_InputPLC;
	stRotaryTransferTorqueLimiter		: ST_IO2_InputPLC;
	stRotaryTransferDelayStop1			: ST_IO2_InputPLC;
	stRotaryTransferDelayStop2			: ST_IO2_InputPLC;

	stLoweratorGuideRHLowerInPosition	: ST_IO2_InputPLC;
	stLoweratorGuideLHLowerInPosition	: ST_IO2_InputPLC;

	stAdditionalConveyor1Isolator		: ST_IO2_InputPLC;
	stAdditionalConveyor2Isolator		: ST_IO2_InputPLC;
	stAdditionalConveyor3Isolator		: ST_IO2_InputPLC;
	stAdditionalConveyor4Isolator		: ST_IO2_InputPLC;

	stAdditionalConveyor4OK				: ST_IO2_InputPLC;

	stConveyorIndexContact				: ST_IO2_InputPLC;

(*METS SADDLE (Gating&Reject System) Filtered Inputs  FB***************************************************************************************************************)

	stOuterAtClamp						: ST_IO2_InputPLC;
	stOuterAtLabelGate					: ST_IO2_InputPLC;
	stSaddlePressureOK					: ST_IO2_InputPLC;
	stGateImpactSensor					: ST_IO2_InputPLC;
	stGateClear							: ST_IO2_InputPLC;


(*METS PLAS Machine Filtered Inputs ***************************************************************************************************************)
	(*Wrapper*)
	
	stMasterlistDoorGuard1				: ST_IO2_InputPLC;
	stMasterlistDoorGuard2				: ST_IO2_InputPLC;
	stMasterlistDoorGuard3				: ST_IO2_InputPLC;

	stOuterBrushOpen					: ST_IO2_InputPLC;
	stPackAggregationDoorGuard1			: ST_IO2_InputPLC;
	stPackAggregationDoorGuard2			: ST_IO2_InputPLC;

	stWrapperDoorGuard1					: ST_IO2_InputPLC;
	stWrapperDoorGuard2					: ST_IO2_InputPLC;

	stHeatTunelPackReject				: ST_IO2_InputPLC;
	stWrapperPackReject					: ST_IO2_InputPLC;
	stWrapperPackReject2				: ST_IO2_InputPLC;
	stWrapperOuterComplete				: ST_IO2_InputPLC;

	stInhibitIntermediateCamera			: ST_IO2_InputPLC;
	stFilmInPosition					: ST_IO2_InputPLC;
	stIntermediatePrinterTrigger		: ST_IO2_InputPLC;

(*METS Labellers Filtered Inputs ***************************************************************************************************************)

	stLabeller1InPosition				: ST_IO2_InputPLC;
	stLabeller1OuterAtLabeller			: ST_IO2_InputPLC;

	stLabeller1Ready					: ST_IO2_InputPLC;
	stLabeller1DataReady				: ST_IO2_InputPLC;
	stLabeller1HomePosition				: ST_IO2_InputPLC;
	stLabeller1LabelPrinted				: ST_IO2_InputPLC;
	stLabeller1ReadyToApply				: ST_IO2_InputPLC;
	stLabeller1ApplyDone				: ST_IO2_InputPLC;
	stLabeller1SummaryWarning			: ST_IO2_InputPLC;
	stLabeller1Error					: ST_IO2_InputPLC;

	stLabeller2InPosition				: ST_IO2_InputPLC;
	stLabeller2OuterAtLabeller			: ST_IO2_InputPLC;

	stLabeller2Ready					: ST_IO2_InputPLC;
	stLabeller2DataReady				: ST_IO2_InputPLC;
	stLabeller2HomePosition				: ST_IO2_InputPLC;
	stLabeller2LabelPrinted				: ST_IO2_InputPLC;
	stLabeller2ReadyToApply				: ST_IO2_InputPLC;
	stLabeller2ApplyDone				: ST_IO2_InputPLC;
	stLabeller2SummaryWarning			: ST_IO2_InputPLC;
	stLabeller2Error					: ST_IO2_InputPLC;

(*METS PAOL  Filtered Inputs ***************************************************************************************************************)

	stPreMachineBuildBack			: ST_IO2_InputPLC;
	stTPDExitBlocked				: ST_IO2_InputPLC;
	(*stInfeedConveyorStart			: ST_IO2_InputPLC;*)

	stPackSeparationDriveOK			: ST_IO2_InputPLC;
	stInfeedConveyorDriveOK			: ST_IO2_InputPLC;

	stPackAggregCameraRigSensor		: ST_IO2_InputPLC;
(*	stPackAggregCameraTrig1Sensor	: ST_IO2_InputPLC;
	stPackAggregCameraTrig2Sensor	: ST_IO2_InputPLC;
	stPackAggregCameraTrig3Sensor	: ST_IO2_InputPLC;
	stPackAggregCameraTrig4Sensor	: ST_IO2_InputPLC;*)

	stPackIsolatorDrive				: ST_IO2_InputPLC;

(*METS General Outputs  ***************************************************************************************************************)

	stSafetyResetSignal				: ST_IO2_OutputPLC;
	stAdditionalSafetyResetSignal	: ST_IO2_OutputPLC;
	stResetPBIndicator				: ST_IO2_OutputPLC;

(*METS TPD Outputs ***************************************************************************************************************)

	stTPDMachineRun				: ST_IO2_OutputPLC;
	stCMLConvoyerRun			: ST_IO2_OutputPLC;
	stEUCAPreMachineRun			: ST_IO2_OutputPLC;
	stEUCAMachineRun			: ST_IO2_OutputPLC;

	stOuterValidationOK			: ST_IO2_OutputPLC;
	stCaseContentOK				: ST_IO2_OutputPLC;
	stCaseValidationOK			: ST_IO2_OutputPLC;
	stLabellerInhibit			: ST_IO2_OutputPLC;

	stPackAggregCamLensAir		: ST_IO2_OutputPLC;
	(*stOuterRejetct				:	ST_IO2_OutputPLC;
	stMLCameraLightning			:	ST_IO2_OutputPLC;
	stAggCameraLightning		:	ST_IO2_OutputPLC;
	stConfCameraLightning		:	ST_IO2_OutputPLC;
	stOuterAggCameraLightning	:	ST_IO2_OutputPLC;*)

(*METS Camera Filtered Outputs ***************************************************************************************************************)

	aCameraOutput				: ARRAY[1..cMAX_CAMERA_NUMBER] OF ST_IO2_OutputPLC;	(**)

	(*stCamera01Out				:	ST_IO2_OutputPLC;
	stCamera02Out				:	ST_IO2_OutputPLC;
	stCamera03Out				:	ST_IO2_OutputPLC;
	stCamera04Out				:	ST_IO2_OutputPLC;
	stCamera05Out				:	ST_IO2_OutputPLC;
	stCamera06Out				:	ST_IO2_OutputPLC;
	stCamera07Out				:	ST_IO2_OutputPLC;
	stCamera08Out				:	ST_IO2_OutputPLC;
	stCamera09Out				:	ST_IO2_OutputPLC;
	stCamera10Out				:	ST_IO2_OutputPLC;
	stCamera11Out				:	ST_IO2_OutputPLC;
	stCamera12Out				:	ST_IO2_OutputPLC;*)


	aCameraLightning			: ARRAY[1..cMAX_CAMERA_NUMBER] OF ST_IO2_OutputPLC;	(**)

	(*stCamera01Lightning				:	ST_IO2_OutputPLC;
	stCamera02Lightning				:	ST_IO2_OutputPLC;
	stCamera03Lightning				:	ST_IO2_OutputPLC;
	stCamera04Lightning				:	ST_IO2_OutputPLC;
	stCamera05Lightning				:	ST_IO2_OutputPLC;
	stCamera06Lightning				:	ST_IO2_OutputPLC;
	stCamera07Lightning				:	ST_IO2_OutputPLC;
	stCamera08Lightning				:	ST_IO2_OutputPLC;
	stCamera09Lightning				:	ST_IO2_OutputPLC;
	stCamera10Lightning				:	ST_IO2_OutputPLC;
	stCamera11Lightning				:	ST_IO2_OutputPLC;
	stCamera12Lightning				:	ST_IO2_OutputPLC;*)

(*METS LightPole Filtered Outputs ***************************************************************************************************************)

	stLightPoleGreen				: ST_IO2_OutputPLC;		(**)
	stLightPoleAmber				: ST_IO2_OutputPLC;		(**)
	stLightPoleRed					: ST_IO2_OutputPLC;		(**)
	stLightPoleAlarm				: ST_IO2_OutputPLC;		(**)
	stHandScannerGreen				: ST_IO2_OutputPLC;		(**)
	stHandScannerRed				: ST_IO2_OutputPLC;		(**)
	stGreenButtonLamp				: ST_IO2_OutputPLC;		(**)

(*METS Drives Filtered Outputs ***************************************************************************************************************)

	stDriveFaultAcknowledge		: ST_IO2_OutputPLC;		(**)
	
	stSideBeltDriveBrake		: ST_IO2_OutputPLC;		(**)
	stInfeedConveyorDriveRun	: ST_IO2_OutputPLC;

	stPackSeparatorDriveBrake	: ST_IO2_OutputPLC;		(**)
	stPackSeparationDriveRun	: ST_IO2_OutputPLC;

	stAdditionalConveyor1Run	: ST_IO2_OutputPLC;
	stAdditionalConveyor2Run	: ST_IO2_OutputPLC;
	stAdditionalConveyor3Run	: ST_IO2_OutputPLC;
	stAdditionalConveyor4Run	: ST_IO2_OutputPLC;

(*METS Cylinders Filtered Outputs ***************************************************************************************************************)

	stClampCylinderExtend				: ST_IO2_OutputPLC;		(**)
	stClampCylinderRetract				: ST_IO2_OutputPLC;

	stGateCylinderExtend				: ST_IO2_OutputPLC;		(**)
	stGateCylinderRetract				: ST_IO2_OutputPLC;

	stRejectCylinderExtend				: ST_IO2_OutputPLC;		(**)
	stRejectCylinderRetract				: ST_IO2_OutputPLC;

	stAdditionalRejectCylinderExtend	: ST_IO2_OutputPLC;		(**)
	stAdditionalRejectCylinderRetract	: ST_IO2_OutputPLC;

	stFirstPusherCylinderExtend			: ST_IO2_OutputPLC;		(**)
	stFirstPusherCylinderRetract		: ST_IO2_OutputPLC;

	stSecondPusherCylinderExtend		: ST_IO2_OutputPLC;		(**)
	stSecondPusherCylinderRetract		: ST_IO2_OutputPLC;

	stRejectActiveNCW					: ST_IO2_OutputPLC;

(*METS Printers Filtered Outputs ***************************************************************************************************************)

	stLabeller1Reset					: ST_IO2_OutputPLC;
	stLabeller1Print					: ST_IO2_OutputPLC;
	stWhiteLabe11Print					: ST_IO2_OutputPLC;
	stLabeller1Apply					: ST_IO2_OutputPLC;
	stLabbeller1ApplyAvailable			: ST_IO2_OutputPLC;

	stLabeller2Reset					: ST_IO2_OutputPLC;
	stLabeller2Print					: ST_IO2_OutputPLC;
	stWhiteLabe12Print					: ST_IO2_OutputPLC;
	stLabeller2Apply					: ST_IO2_OutputPLC;
	stLabbeller2ApplyAvailable			: ST_IO2_OutputPLC;

	stIntermediatePrinterTrigger1		: ST_IO2_OutputPLC;

(*METS Laser Filtered Outputs ***************************************************************************************************************)

	stLaserEnable						: ST_IO2_OutputPLC;
	stLaserPrintAllow					: ST_IO2_OutputPLC;
	stPrintStart						: ST_IO2_OutputPLC;	

END_VAR

// ---- Global Variables/gPersistent.TcGVL
{attribute 'qualified_only'}
{attribute 'Tc2GvlVarNames'}
VAR_GLOBAL PERSISTENT

(**************************************************************************************************************)
(* Local persistend data, not important currently form METS process perspective, but not removed to keep consistency		*)
(* with old version of software.																		*)
(**************************************************************************************************************)
	stWriteOCVFileStatistic			: ST_FILE_WriteFileStatistic;
	stWriteOACFileStatistic			: ST_FILE_WriteFileStatistic;	(*Move to METSEfficency one day*)
	stWriteCHMFileStatistic			: ST_FILE_WriteFileStatistic;	(*Move to METSEfficency one day*)

	stLocalCHMData					: ST_CHM_Data;	(* CHM data printed to XML file *)

	bRefreshSystemIno				: BOOL;

	nReadOCVError					: UDINT;
	nReadOCVFound					: UDINT;
	nReadOCVFoundInErr				: UDINT;

	nValidationTrigerMonitroing 	: UINT;
	tValidationTrigerTimeout		: TIME :=t#5000ms;

	nAirPrssureMonitoring			: UINT;
	tAirPressureTimeout				: TIME :=T#5000MS;

	nPrinterHomeMonitoring			: UINT;
	tPrinterHomeTimeout				: TIME :=T#5000MS;

	nGateRetractMonitoring			: UINT;
	tGateRetractTimeout				: TIME :=T#5000MS;

	nCasHeadCounter					: UDINT;
	nOuterHeadCounter				: UDINT;
	nCaseEndCounter					: UDINT;

	bEnableSUPICheck				: BOOL;	 	(*Enable SUPI check for pack code*)
	nSUPI_Identyfication			: DINT;

	(*pack code validation*)
	nPackCodeTooShortIndex			: UDINT;	(*READ*)
	nPackCodeTooLongIndex			: UDINT;	(*READ*)
	nPackCodeTypeErrorIndex			: UDINT;	(*READ*)

	nRestoredOCVSuccessful			: UDINT;	(*READ*)
	nRestoredOCVProcessed			: UDINT;	(*READ*)

	bDisableInfeedQueueAlarm 		: BOOL;
	bDisablePackerQueueAlarm		: BOOL;

	sLastFileNameToDlogHMI			: T_CAC_Filename;	(*READ/WRITE BY HMI ONLY*)
	sLastFileTimeToDlogHMI			: STRING(19);		(*READ/WRITE BY HMI ONLY*)

	nStackIndexDebug				: ARRAY[0..10] OF UDINT;
	
	nRecoverOuterLable				: INT;

	(*sHMICaseStats				 	: ST_SCANNER_Statistics;*)

(*	fbShiftPackMonitor	: FB_KPI_ChangeItemsProducedTrig;
	fbShiftOuterMonitor	: FB_KPI_ChangeItemsProducedTrig;
	fbShiftCaseMonitor	: FB_KPI_ChangeItemsProducedTrig;
	fbProdPackMonitor	: FB_KPI_ChangeItemsProducedTrig;
	fbProdOuterMonitor	: FB_KPI_ChangeItemsProducedTrig;
	fbProdCaseMonitor	: FB_KPI_ChangeItemsProducedTrig;*)

	stEmptyEfficiency				: ST_NOVRAM_METS_Inspection;

	strLastBarcodeRead				: STRING(255);
	tPassthroughDelay				: TIME := T#180MS;

	(*strHMIVersionInfo				: STRING;
	strPLCVersion					: STRING;
	strPLCVersionInfo				: STRING;
*)
	nWriteOCVErrorIndex			: UINT;
	nWriteOACErrorIndex			: UINT;
	nReadOCVErrorIndex			: UINT;


	bEUCAMonitorEthernet		: BOOL := FALSE;
	bTPDMonitorEthernet			: BOOL := FALSE;
	bEUCAAirConditionExist		: BOOL := FALSE;
	bTPDAirConditionExist		: BOOL := FALSE;

	(*sCameraPack				: ARRAY[1..6] OF ST_SCANNER; 	(*PACK AGGREGATION OR INTERMEDIAT CAMERAs*)*)

	bUseMultipleOuterFormats		: BOOL := FALSE;
	bInfeedRejectFitted				: BOOL;

	bCaseValidationOverTime 		: BOOL;
END_VAR

// ---- Global Variables/gNovRAM.TcGVL
{attribute 'qualified_only'}
{attribute 'Tc2GvlVarNames'}
VAR_GLOBAL

(* *********************************************************** *)
(* *********    Non-volatile data    CASE PACKER     ********* *)
(* *********************************************************** *)
(* Non-volatile data - for CX2030, the CPU has a 128 kB (up to %MB131072 ) NOVRAM persistent data memory for situations where no UPS is used. *)

	bInitBit							AT %MX0.0 		: BOOL := TRUE; 					(* must not be moved *)

	stMetsCamerasNV						AT %MB8			: ST_NOVRAM_METS_Cameras;			(*Size 811 B - allocated 999 B*)
	stMetsEfficiencyNV					AT %MB1000		: ST_NOVRAM_METS_Inspection; 		(*Size 515 B  - allocated 600 B*)
	stCasePackerSignalsNV				AT %MB1600		: ST_NOVRAM_METS_DualInputs;		(*Size 103 B - allocated 150 B*)
	stCaseInspactionLogNV				AT %MB1748		: ST_NOVRAM_METS_CaseInspactionLog;	(*Size 115 B  - allocated 150 B*)

	sCurrentCHMArchiveDateNameNV		AT %MB1900		: STRING(11);						(*Size 12 B  - allocated 20 B*)
	sNewCHMArchiveDateNameNV			AT %MB1920		: STRING(11);						(*Size 12 B  - allocated 20 B*)
	sLastSendingTimeToFactoryLayerNV	AT %MB1940		: STRING(19);						(*Size 20 B  - allocated 20 B*)
	(*nDummySecquentionalCounter		AT %MB1960		: UDINT;*)							(*Size 8 B  - allocated 20 B*)

	stShiftStatisticNV					AT %MB2000		: ST_NOVRAM_METS_EventCounters; 	(*Size 14597 B - allocated 15000 B*)
	stProdStatisticNV					AT %MB17000		: ST_NOVRAM_METS_EventCounters; 	(*Size 14597 B - allocated 15000 B*)

	nNVChecksum							AT %MB32764	: WORD;									(* must not be moved *)

END_VAR

// ---- Global Variables/METS/gDevice.TcGVL
{attribute 'qualified_only'}
{attribute 'Tc2GvlVarNames'}
VAR_GLOBAL
	
(**************************************************************************************************************)
(* Global structures or variables, releted to general METS proces form perspectiv of EUCA unit. 						*)
(* Outer to case aggregation proccess																	*)
(**************************************************************************************************************)

(* *********************************************************** *)
(**********Core METS  state and configuration structures************)
(* *********************************************************** *)
	eMachineState						: E_SYSTEM_MachineState;
	stMachineState						: ST_SYSTEM_MachineState;
	sActiveMachineState					: STRING; 
	
	bForceMachineState					: BOOL := FALSE;
	nForcedMachineState					: INT;
	
	stMetsStatus						: ST_SYSTEM_MachineStatus;
	stMachineConfig						: ST_SYSTEM_Config;
	stMachineSafety						: ST_SYSTEM_SafetyStatus;
	stMachineDevices					: ST_SYSTEM_DeviceState;
	
	eAutomationMode						: E_SYSTEM_AutomationMode;
	
(* *********************************************************** *)
(* ***************        Genreal PLC section	 ************************)
(* *********************************************************** *)

	stEtherCATStatus					: ST_EtherCATStatus;
	
	fbXFastTaskkInfo					: FB_SYSTEM_TaskInfo;
	stXFastTaskSys						: PlcTaskSystemInfo;
	bXFastTask1stCycle					: BOOL;
	tXFastTaskCycleTime					: TIME;
	
	fbFastTaskkInfo						: FB_SYSTEM_TaskInfo;
	stFastTaskSys						: PlcTaskSystemInfo;
	bFastTask1stCycle					: BOOL;
	tFastTaskCycleTime					: TIME;
	
	fbControlTaskInfo					: FB_SYSTEM_TaskInfo;
	stControlTaskSys					: PlcTaskSystemInfo;
	bControlTask1stCycle				: BOOL;
	tControlCycleTime					: TIME;

	fbAuxTaskInfo						: FB_SYSTEM_TaskInfo;
	stAuxTaskSys						: PlcTaskSystemInfo;
	bAuxTask1stCycle					: BOOL;
	tAuxCycleTime						: TIME;
	
	stPLCAppSys							:	PlcAppSystemInfo;

	bProductInstructionValid			: BOOL;
	
	
(* *********************************************************** *)
(* ****************        DB section	 ******************************)
(* *********************************************************** *)

	(*stCACCheck						: ST_DB_CACCheckCtrl;*)
	stDBReport							: ST_DB_ReportDBCtrl;
	
(* *********************************************************** *)
(* ****************       Pulse signal	 **************************)
(* *********************************************************** *)

	bPulse05s							: BOOL;
	bPulse1s							: BOOL;
	bPulse2s							: BOOL;
	bPulse5s							: BOOL;	
	bPulse10s							: BOOL;
	
(* ************************************************************)
(* ******************       Bridge 	 *************************)
(* ************************************************************)

	stBridge							: ST_SYSTEM_BridgeStatus;
	nWatchdogToBridge					: DINT;
	nWatchdogFromBridge					: DINT;


(* *********************************************************** *)
(* ******************       Logger 	 **************************)
(* *********************************************************** *)

	stProcessLogger						: ST_SYSTEM_LoggerStatus;
	nWatchdogToLogger					: DINT;
	nWatchdogFromLogger					: DINT;
	

(* *********************************************************** *)
(* ******************       DB 	 **************************)
(* *********************************************************** *)

	stArchiveDB							: ST_SYSTEM_ArchiveDBStatus	;
	nWatchdogToArchiveDB				: DINT;
	nWatchdogFromArchiveDB				: DINT;

(* *********************************************************** *)
(* ***************     Reporting  KPI	 ***********************)
(* *********************************************************** *)

	stReportingDB						: ST_SYSTEM_ReportingDBStatus	;
	nWatchdogToReportingDB				: DINT;
	nWatchdogFromReportingDB			: DINT;

(* *********************************************************** *)
(* ****************       Cameras  ******************************)
(* *********************************************************** *)

	aCameraControl						: ARRAY[1..cMAX_CAMERA_NUMBER] OF ST_SCANNER_CameraMap;
	aCameraLightingIntensity			: ARRAY[1..cMAX_CAMERA_NUMBER] OF INT;

	nLightboxLightingIntensityTop		: INT;	(*use as all*)
	nLightboxLightingIntensityBottom	: INT; (*ue in METS ONE*)

	(*nPackAggregationLightingIntensity		: INT;
	nPackConfirmationLightingIntensity		: INT;
	nMasterlistCameraLightingIntensity		:INT;*)

(* *********************************************************** *)
(* ****************       Profinet	 ******************************)
(* *********************************************************** *)

	aG120Control						: ARRAY[1..cMAX_PROFINET_DRIVES] OF ST_G120_Control;

(* *********************************************************** *)
(* ****************       Cylinders	 ******************************)
(* *********************************************************** *)

	aCylinderControl					: ARRAY[1..cMAX_CYLINDERS] OF ST_CYLINDER_Control;

(* *********************************************************** *)
(* ****************      Axis	 ******************************)
(* *********************************************************** *)


	aAxisControl						: ARRAY[1..cMAX_MC2_DRIVES] OF ST_AXIS_Control;
	aAxisParamSet						: ARRAY[1..cMAX_MC2_DRIVES] OF ST_AxisParameterSet;

(* *********************************************************** *)
(* ****************       Printers	 ******************************)
(* *********************************************************** *)

	aSecquentionalCounter				: ARRAY[1..cMAX_PRINTER_NUMBER] OF UDINT;
	nDummySecquentionalCounter			: UDINT;


END_VAR

// ---- Global Variables/METS/gProcess.TcGVL
{attribute 'qualified_only'}
{attribute 'Tc2GvlVarNames'}
VAR_GLOBAL
(**************************************************************************************************************)
(* Global structures or variables, releted to general METS proces form perspectiv of TPD unit.	 						*)
(* Pack to outer aggregation proccess																	*)
(**************************************************************************************************************)
(* *********************************************************** *)
(************   Core TPD pack aggregation structures 	************)
(* *********************************************************** *)

	ePackAggregationMode				: E_SYSTEM_PackAggregationMode;
	eOuterAggregationMode				: E_SYSTEM_OuterAggregationMode;

	aPackSecondaryMasterListQueue		: ARRAY[1..cMAX_PACK_INFEED_QUEUE] OF ST_PACK_Data; (* Refeed queue *)
	aPackPrimaryMasterListQueue			: ARRAY[1..cMAX_PACK_INFEED_QUEUE] OF ST_PACK_Data; (* Refeed queue *)

	(*aPackTracingQueue					: ARRAY[1..cMAX_TRACE_UNIT_QUEUE] OF ST_PACK_Data;
	aPackRejectedQueue					: ARRAY[1..cMAX_PACK_REJECTED_QUEUE] OF ST_PACK_Data;*)
	(*stPackInTransferQueue					: ST_PACK_InfeedQueue; (*Stacker queu*)*)

	stPackInfeedQueue					: ST_PACK_InfeedQueue; (* Infeed queue *)
	aMultiPackInfeedQueue				: ARRAY[1..cMAX_CAMERA_PROG_NUMBER] OF ST_PACK_InfeedQueue;

	aStackerQueue							: ARRAY[1..cMAX_PACK_INFEED_QUEUE] OF ST_PACK_Data;

	aLastFilledCodes						: ARRAY[1..cMAX_PACK_INFEED_QUEUE] OF ST_PACK_LastFilledCodes;

	aInterimCodeQueue					: ARRAY[1..cMAX_INTERMEDIATE_CODE_QUEUE] OF T_MaxString;

	aOCVPackStatus						: ARRAY[1..cMAX_OUTER_STATUS_QUEUE] OF ST_OUTER_Status;	(* Outer status register - would be nice to call it PACK Status and remove unnecesary stuff*)
	stLastOCVStatus						: ST_OUTER_Status;
	aErrorOCVPack							: ARRAY[1..cMAX_OUTER_STATUS_QUEUE] OF ST_OUTER_Status;
	stErrorOCVPack						: ST_OUTER_Status;

	stCurrentOuterStatus					: ST_OUTER_Status;	(* Outer status *)
	aOuterStatus							: ARRAY[1..cMAX_OUTER_STATUS_QUEUE] OF ST_OUTER_Status;	(* Outer status register *)
	stLastOuterStatus						: ST_OUTER_Status;
	aErrorOuters							: ARRAY[1..cMAX_OUTER_STATUS_QUEUE] OF ST_OUTER_Status;
	stErrorOuter							: ST_OUTER_Status;



(* *********************************************************** *)
(* *********      LARS  - evaluation  ************************)
(* *********************************************************** *)

	(*bRejectNotConfirmed	: BOOL;*)

(* *********************************************************** *)
(* *********      Side Flex  - evaluation  ************************)
(* *********************************************************** *)

	bSideFlexInitRun					: BOOL;
	bSideFlexPackToOuterProcessing	: BOOL;

	stSideFlexProcessData					: ST_SIDEFLEX_ProcessData;

	(*bSideFlexAggCameraTrigger	: BOOL;

	bSideFlexTwoOuterInAggregationArea	: BOOL;
	bSideFlexRejectNotConfirmed	: BOOL;
	bSideFlexTransferNotConfirmed	: BOOL;
	bSideFlexOuterAtChuteExitNotConfirmed	: BOOL;*)


	(*bInputSensor					: BOOL;
	aProcessData					: ARRAY[1..cMAX_SIDEFLEX_QUEUE] OF ST_SIDEFLEX_ProcessData;
	aConvrStatusUpdate			: ARRAY[1..cMAX_SIDEFLEX_QUEUE] OF FB_SIDEFLEX_ConvStatusUpdate;
	stSideFlexOffset				: ST_SIDEFLEX_Offset;
	nValidationIndexPointer		: INT;
	bSideFlexApplyLabel			: BOOL;
	bSideFlexOuterValidationTrig	: BOOL;*)


(* *********************************************************** *)
(* ******************       DB 	 **************************)
(* *********************************************************** *)

	aOCVDataDB	: ARRAY[0..7] OF	ST_DB_OCVDataCtrl;
	aOACDataDB	: ARRAY[0..6] OF	ST_DB_OACDataCtrl;
	aCACDataDB	: ARRAY[0..5] OF	ST_DB_CACDataCtrl;

(* *********************************************************** *)
(* *********       Log  ************************)
(* *********************************************************** *)
	aLogHandler				: ARRAY[0..255] OF FB_LOG_Handler;

	stEventDataPT				: ST_LOG_EventData;
	stEventDataML				: ST_LOG_EventData;
	stEventDataOT				: ST_LOG_EventData;
	stEventDataCT				: ST_LOG_EventData;

	stWriteImageData			: ST_LOG_WriteImageData;

(* *********************************************************** *)
(* *********      File write error  ************************)
(* *********************************************************** *)
	aLogOCVFileWriteError		: ARRAY[1..10] OF ST_LOG_FileWriteError;
	aLogOACFileWriteError		: ARRAY[1..10] OF ST_LOG_FileWriteError;
	aLogCACFileWriteError		: ARRAY[1..10] OF ST_LOG_FileWriteError;
	aLogCHMFileWriteError		: ARRAY[1..10] OF ST_LOG_FileWriteError;

(* *********************************************************** *)
(* *********        Core Structures for EUCA ************************)
(* *********************************************************** *)

	aOuterMasterListQueue					: ARRAY[0..cMAX_OUTER_STATUS_QUEUE] OF T_MaxString;
	stOrcaData							: ST_ORCA_Data;
	stInfeedConvQueue						: ST_CASE_InfeedQueue;

	aPackerQueue							: ARRAY [0..1] OF ST_CASE_InfeedQueue;
	stCaseQueue							: ST_CASE_CaseQueue;

	bManualCaseScan						: BOOL;
	aFailedCACData						: ARRAY[1..cMAX_FAILED_CASE_QUEUE] OF ST_CAC_Data;	(* array of failed CAC data *)
	aVerifiedCACData						: ARRAY[1..cMAX_VERIFIED_CASE_QUEUE] OF ST_CAC_Data;	(* array of verified CAC data *)


(* *********************************************************** *)
(* ***************       Clear queue by door section	 ************************)
(* *********************************************************** *)

	stDoorOpenClearData					: ST_SYSTEM_Door;
	bClearConveyorQueue					: BOOL;
	bClearPackerQueue						: BOOL;
	bClearCaseQueue						: BOOL;

(* *********************************************************** *)
(* ***************        MasterList section	 ************************)
(* *********************************************************** *)

	bMasterListBarcodeAdded				: BOOL;
	bMasterListCheckComplete				: BOOL;
	nMasterListRestoreCounter				: INT;			(*number of restored Outers in one case*)

(* *********************************************************** *)
(* ***************        Validation section	 ************************)
(* *********************************************************** *)

	

	stPackRejectReasons					: ST_RejectReasonsForPack;
	stOuterRejectReasons					: ST_RejectReasonsForOuter;
	stCaseRejectReasons					: ST_RejectReasonsForCase;

	aRejectCountersID						: ARRAY[0..cMAX_REJECT_REASON] OF UINT;

	(*bSetOuterValidationOK				: BOOL;
	bSetOuterValidationNOK				: BOOL;*)
	bSetEarlyCaseValidationOK			: BOOL;
	bSetEarlyCaseValidationNOK			: BOOL;
	bSetCaseValidationOK					: BOOL;
	bSetCaseValidationNOK				: BOOL;
	bInhibitPulseAlarmOK					: BOOL;
	bSetPulseAlarmNOK					: BOOL;


(* *********************************************************** *)
(* ***************     Pack aggregation  **************************)
(* *********************************************************** *)

	bPackInfeedConveyerIsRuning				: BOOL;
	bRunSeparationDrive					: BOOL;
	bOuterInsideLighBox					: BOOL;
	bOuterInsideRotartyPosition				: BOOL;
	bCamerasOutOfSync						: BOOL;
	bInhibitPackSeparator_CameraBufferHigh	: BOOL;

	bIncrementAggregationFIFO				: BOOL;
	bFillInAggregationFIFO					: BOOL;

(*	bTPDCutOutFromConv					: BOOL;
	bTPDCutOutFromSeparator				: BOOL;*)

	nPackNoReadCounter					: INT;

	bAddToPackMLQueueDone				: BOOL;
	bAddToPackQueueDone					: BOOL;
	bAddToStackerQueueDone				: BOOL;
	bAddToInterimQueueDone					: BOOL;

(* *********************************************************** *)
(* ***************     Outer aggregation  **************************)
(* *********************************************************** *)

	bSearchCode							: BOOL;
	sNewPackCodeRefeed					: T_PACK_Barcode;

	nOuterNoReadCounter					: INT;

	(*bManualInterimCodeTrigger				: BOOL;*)
	stManualInterimImageData				: ST_SCANNER_ImageData;					(*f.ex can by used F21_HandScanner.strCaseBarcode*)

	nOuterCounterValue					: UINT;

	bValidateForRejectDone				: BOOL;
	bValidateForRejectBusy				: BOOL;
	bValidateForRejectError				: BOOL;
	nValidateForRejectErrorID				: UDINT;

	bRejectCurrentOuter					: BOOL := TRUE;
	sCurrentOuterRejectCode				: STRING(255);

	(*bManualOuterLabelEnable				: BOOL;*)
	bManualOuterLableTrigger				: BOOL;
	sManualOuterLabelBarcode			: T_OUTER_Barcode;					(*f.ex can by used F21_HandScanner.strCaseBarcode*)

	stCurrentPackerData					: ST_CASE_OperationData;

	(*bManualRowLabelEnable					: BOOL;*)
	bManualRowLableTrigger					: BOOL;
	sManualRowLabelBarcode					: T_OUTER_Barcode;					(*f.ex can by used F21_HandScanner.strCaseBarcode*)

	stOuterPrintStationStruct					: ST_OuterPrintStationStruct;

(* *********************************************************** *)
(* ***************        Case aggregation	 ************************)
(* *********************************************************** *)
	bOuterRemovedFromInfeedQueue			: BOOL;
	bWaitingCaseContentRead				: BOOL;
	bWaitngCaseDischarge					: BOOL;
	bCaseDischargeExecution					: BOOL;
	bWaitingToScanLabel					: BOOL;
	bResetForWaitingScanCaseLable			: BOOL;
	bCaseRejectedBeforeScanLabelSignal 		: BOOL;

	(*bManualCaseLabelEnable					: BOOL;*)
	bManualCaseLableTrigger					: BOOL;
	sManualCaseLabelBarcode				: T_CASE_Barcode;					(*f.ex can by used F21_HandScanner.strCaseBarcode*)

	bORCADataReady						: BOOL;

	sLastCaseLabelBarcode					: T_CASE_Barcode;

	bCaseContetntValidationComplete		: BOOL;
	bCaseValidationOK						: BOOL;					(*Output signal to IO Card - validation OK for casepacker*)
	bCaseValidationNOK						: BOOL;					(*Output signal to IO Card - validation Not OK for casepacker*)

	bCaseValid							: BOOL;
	bCaseInvalid							: BOOL;

(********From Pack Trace variable************************)

	bManualDeleteAllOACFiles				: BOOL;
	bManualDeleteAllOCVFiles				: BOOL;

END_VAR

// ---- Global Variables/_VERSION/_VERSION_CONTROL.TcGVL
{attribute 'Tc2GvlVarNames'}
VAR_GLOBAL
	(*cRELEASE_DATE		: STRING[10] := '25.03.2025';*)

	cHARDWARE_CONFIG_VERSION	: STRING[20] := 'IND-METS-NCW_v007';
	(*cVERSION_INFO		: T_MaxString := '26/07/23 - 07.00.41 - SD - UPS management';*)
END_VAR

(*
Version history:

Date		|	Version/Author 		|	Remark
----------------------------------------------------------------------------------------------------
26/07/23	|	07.00.41	SD		|	UPS management and power related Alarm and Warnings
25/07/23	|	07.00.40	SD		|	UPS management draft
19/07/23	|	07.00.39	SD		|	PLAS sequence placeholder
18/07/23	|	07.00.38	TW SD	|	Hand scsnner selection mod
09/05/23	|	07.00.02	PP		|	Add remaining HotFixes form Korea (according Jira tasks)
			|						|	
09/11/22	|	06.37.05	PP		|	Add Log system for case level (EventCT) and VERSION_CONTROL
05/11/22	|	06.37.03	PP		|	Original PLC-METS-6.37.03_Inline.pro from Piotr
15/09/22	|	06.37.01	PP		|	Lateste hardware design implemented HC METS-INLINE v2.10
*)

// ---- POUs/METS/T01_CONTROL.TcPOU
 PROGRAM T01_CONTROL
VAR
END_VAR

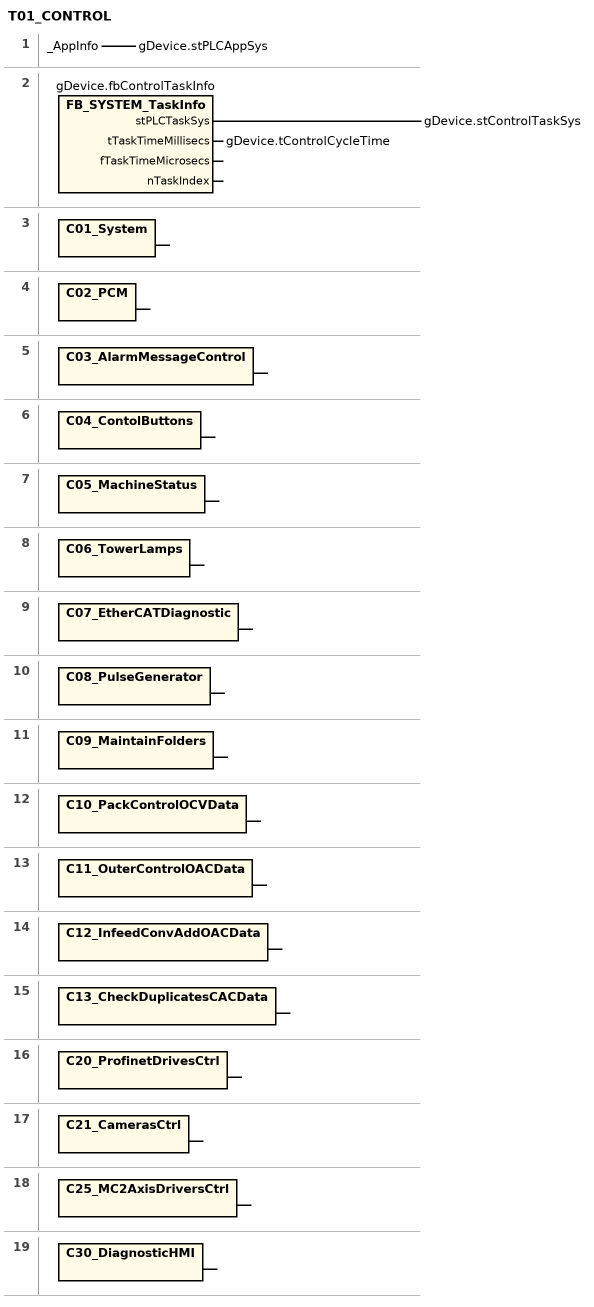
// NETWORK 1
gDevice.stPLCAppSys := _AppInfo;

// NETWORK 2
gDevice.fbControlTaskInfo(tTaskTimeMillisecs => gDevice.tControlCycleTime); // FB_SYSTEM_TaskInfo
gDevice.stControlTaskSys := gDevice.fbControlTaskInfo.stPLCTaskSys;

// NETWORK 3
C01_System();

// NETWORK 4
C02_PCM();

// NETWORK 5
C03_AlarmMessageControl();

// NETWORK 6
C04_ContolButtons();

// NETWORK 7
C05_MachineStatus();

// NETWORK 8
C06_TowerLamps();

// NETWORK 9
C07_EtherCATDiagnostic();

// NETWORK 10
C08_PulseGenerator();

// NETWORK 11
C09_MaintainFolders();

// NETWORK 12
C10_PackControlOCVData();

// NETWORK 13
C11_OuterControlOACData();

// NETWORK 14
C12_InfeedConvAddOACData();

// NETWORK 15
C13_CheckDuplicatesCACData();

// NETWORK 16
C20_ProfinetDrivesCtrl();

// NETWORK 17
C21_CamerasCtrl();

// NETWORK 18
C25_MC2AxisDriversCtrl();

// NETWORK 19
C30_DiagnosticHMI();

END_PROGRAM

// ---- POUs/METS/Common LIB/09_SYSTEM LIB/FB_SYSTEM_TaskInfo.TcPOU
(* task info with times of current task converted to millisecs and microsecs *)
FUNCTION_BLOCK FB_SYSTEM_TaskInfo
VAR_INPUT
END_VAR
VAR_OUTPUT
	stPLCTaskSys		:	PlcTaskSystemInfo;
	tTaskTimeMillisecs	: TIME;		(* Task Time in time format with ms resolution *)
	fTaskTimeMicrosecs	: LREAL;	(* Task Time in LREAL format with us resolution *)
	nTaskIndex			: BYTE;		(* Task Index of task where this FB is called *)
END_VAR
VAR	
	fbGetCurTaskIdx 				: 	GETCURTASKINDEX;
END_VAR
(*
-------------------------------------------------------------------------------------------------
Date		Version	Author	Comments
-------------------------------------------------------------------------------------------------
30/01/2015	3.00.00	PB		No change

-------------------------------------------------------------------------------------------------
15/03/2010	1.01.00	PB		Current PLC Port No added to FB_TaskTime
							bFirstCycle made primary output of FB_TaskTime
05/02/2010	1.00.00	PB		Initial release
							
-------------------------------------------------------------------------------------------------
*)

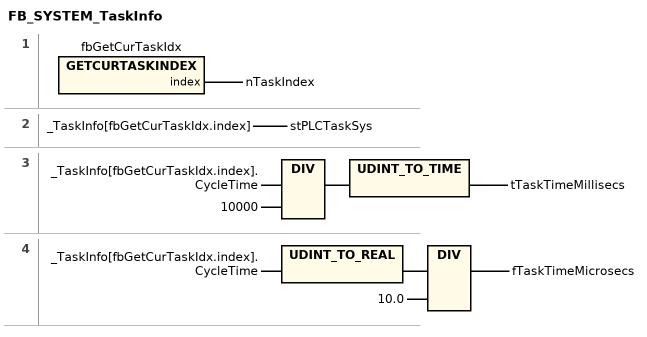
// NETWORK 1
fbGetCurTaskIdx(); // GETCURTASKINDEX
nTaskIndex := fbGetCurTaskIdx.index;

// NETWORK 2
stPLCTaskSys := _TaskInfo[fbGetCurTaskIdx.index];

// NETWORK 3
tTaskTimeMillisecs := UDINT_TO_TIME(_TaskInfo[fbGetCurTaskIdx.index].CycleTime / 10000);

// NETWORK 4
fTaskTimeMicrosecs := UDINT_TO_REAL(_TaskInfo[fbGetCurTaskIdx.index].CycleTime) / 10.0;

END_FUNCTION_BLOCK

// ---- POUs/METS/T03_xFAST.TcPOU
PROGRAM T03_xFAST
VAR
END_VAR

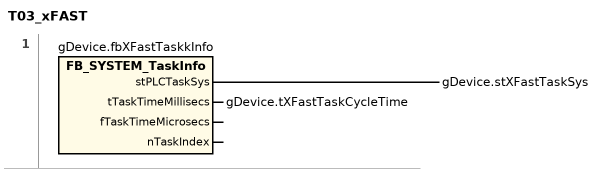
// NETWORK 1
gDevice.fbXFastTaskkInfo(tTaskTimeMillisecs => gDevice.tXFastTaskCycleTime); // FB_SYSTEM_TaskInfo
gDevice.stXFastTaskSys := gDevice.fbXFastTaskkInfo.stPLCTaskSys;

END_PROGRAM

// ---- POUs/METS/T00_FAST.TcPOU
PROGRAM T00_FAST
VAR
	bExecuteDiagnosticBlock	: BOOL;
END_VAR

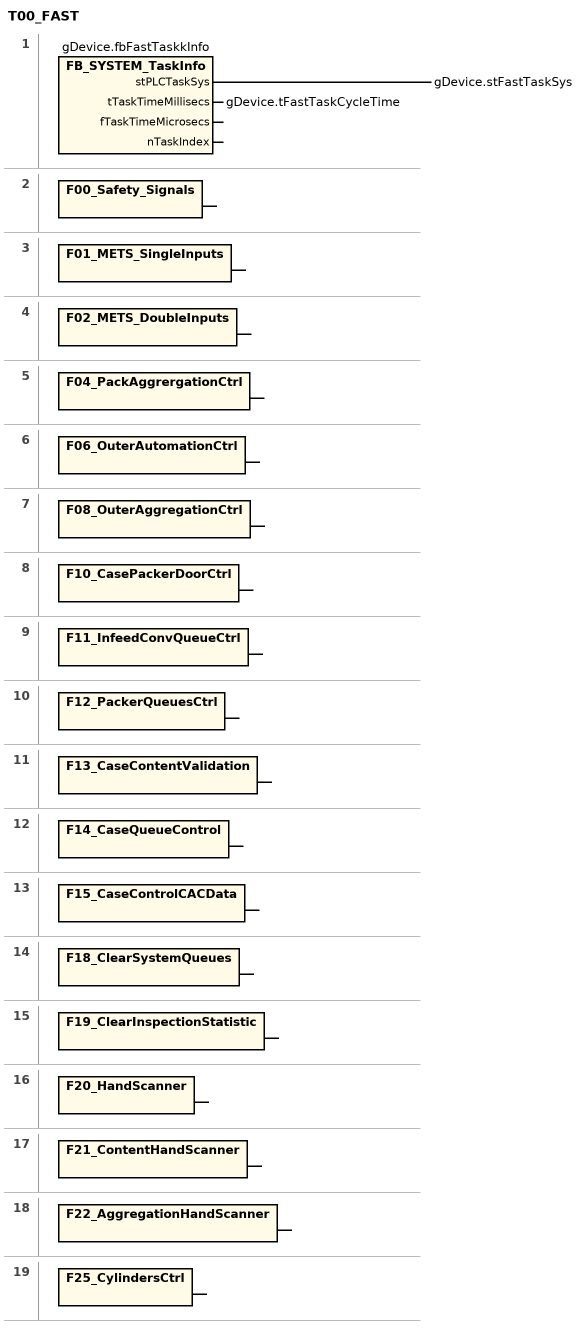
// NETWORK 1
gDevice.fbFastTaskkInfo(tTaskTimeMillisecs => gDevice.tFastTaskCycleTime); // FB_SYSTEM_TaskInfo
gDevice.stFastTaskSys := gDevice.fbFastTaskkInfo.stPLCTaskSys;

// NETWORK 2
F00_Safety_Signals();

// NETWORK 3
F01_METS_SingleInputs();

// NETWORK 4
F02_METS_DoubleInputs();

// NETWORK 5
F04_PackAggrergationCtrl();

// NETWORK 6
F06_OuterAutomationCtrl();

// NETWORK 7
F08_OuterAggregationCtrl();

// NETWORK 8
F10_CasePackerDoorCtrl();

// NETWORK 9
F11_InfeedConvQueueCtrl();

// NETWORK 10
F12_PackerQueuesCtrl();

// NETWORK 11
F13_CaseContentValidation();

// NETWORK 12
F14_CaseQueueControl();

// NETWORK 13
F15_CaseControlCACData();

// NETWORK 14
F18_ClearSystemQueues();

// NETWORK 15
F19_ClearInspectionStatistic();

// NETWORK 16
F20_HandScanner();

// NETWORK 17
F21_ContentHandScanner();

// NETWORK 18
F22_AggregationHandScanner();

// NETWORK 19
F25_CylindersCtrl();

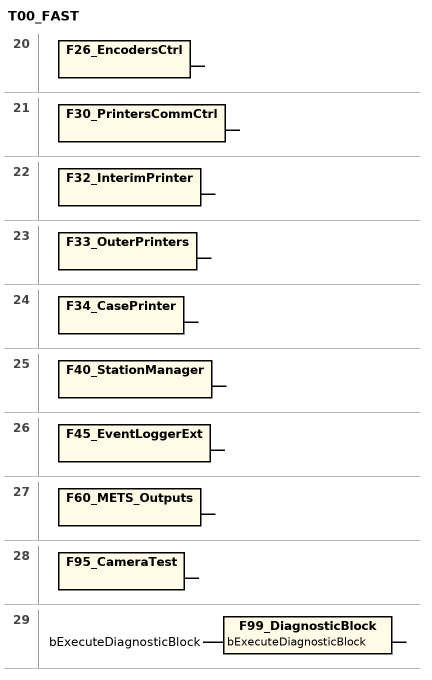
// NETWORK 20
F26_EncodersCtrl();

// NETWORK 21
F30_PrintersCommCtrl();

// NETWORK 22
F32_InterimPrinter();

// NETWORK 23
F33_OuterPrinters();

// NETWORK 24
F34_CasePrinter();

// NETWORK 25
F40_StationManager();

// NETWORK 26
F45_EventLoggerExt();

// NETWORK 27
F60_METS_Outputs();

// NETWORK 28
F95_CameraTest();

// NETWORK 29
F99_DiagnosticBlock(bExecuteDiagnosticBlock := bExecuteDiagnosticBlock);

END_PROGRAM

// ---- POUs/METS/T02_ACCESSORY.TcPOU
PROGRAM T02_ACCESSORY
VAR
END_VAR

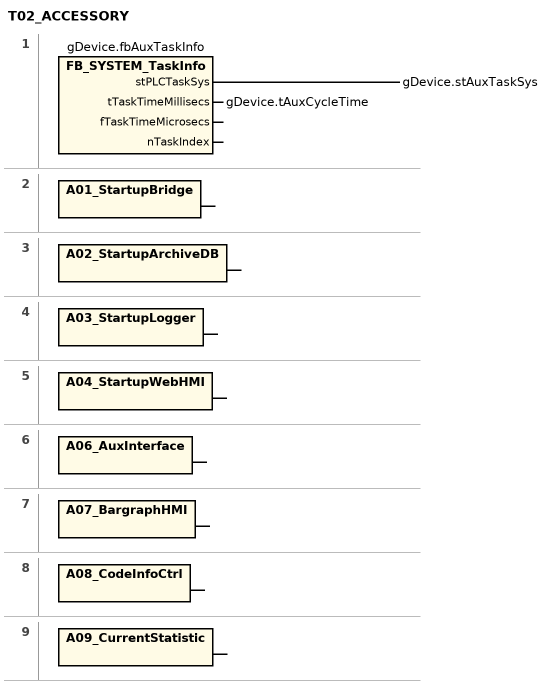
// NETWORK 1
gDevice.fbAuxTaskInfo(tTaskTimeMillisecs => gDevice.tAuxCycleTime); // FB_SYSTEM_TaskInfo
gDevice.stAuxTaskSys := gDevice.fbAuxTaskInfo.stPLCTaskSys;

// NETWORK 2
A01_StartupBridge();

// NETWORK 3
A02_StartupArchiveDB();

// NETWORK 4
A03_StartupLogger();

// NETWORK 5
A04_StartupWebHMI();

// NETWORK 6
A06_AuxInterface();

// NETWORK 7
A07_BargraphHMI();

// NETWORK 8
A08_CodeInfoCtrl();

// NETWORK 9
A09_CurrentStatistic();

END_PROGRAM

// ---- POUs/TcUnit/PRG_TEST.TcPOU
PROGRAM PRG_TEST
VAR
	fbExtractAnyStringTests			: FB_ExtractAnyStringTests;
	fbExtractStringTests			: FB_ExtratcStringTests;
	fbReplaceLongStringCharTests	: FB_ReplaceLongStringCharTests;
	fbLogHandlerTests				: FB_LogHandlerTests;
	
	fbValidateContentTests			: FB_CASE_ValidateContentTests;
END_VAR

//===================================================
//UNIT TEST EXECUTION

TcUnit.RUN();

//===================================================
//MANUAL TEST EXECUTION

PRG_ExtractAnyStringManual();
PRG_ExtractStringManual();
PRG_ReplaceLongSingleCharManual();
PRG_LogHandlerManual();

END_PROGRAM

// ---- POUs/TcUnit/FB_ExtractAnyStringTests/FB_ExtractAnyStringTests.TcPOU
FUNCTION_BLOCK FB_ExtractAnyStringTests EXTENDS FB_TestSuite

//==============================================================
//MAIN TESTS
//==============================================================

testMain01_ModeWITHIDENT_ExactDataNoPurge();
testMain02_ModeWITHIDENTPURGE_ExactDataAndPurge();
testMain03_ModeWITHOUTIDENT_ExtractDataNoPurge();
testMain04_ModeWITHOUTIDENTPURGE_ExtractDataAndPurge();
testMain05_ModeWITHOUTIDENTREMIDENT_ExtractDataNoPurge();
testMain06_ModeWITHOUTIDENTREMIDENTPURGE_ExtractDataAndPurge();
testMain07_ExtractFromLongString_ExtractData();
testMain08_ExtractFromLongString_LenghtExtractedDataOk();
testMain09_ExtractCharOnly_LeftStringWithExtractCharLenght();

//==============================================================
//NEGATIVE TESTS
//==============================================================

testNeg01_ReverseIdentAllModes_EmptyString();
testNeg02_NoSufixFound_EmptyStringNoDataCahnge();
testNeg03_NoPrefixFound_EmptyStringNoDataCahnge();
testNeg04_NoPrefixSufixFoundNoCharsExtr_LeftString();
testNeg05_PrefixFoundNoSufixNoCharsExtr_RightString();

//==============================================================
//SEQUENCE TESTS
//==============================================================

testSeq01_MVxDecode_ImageData();

//==============================================================
//OTHERS TESTS
//==============================================================

//FbExtrctAnyStringTests_ExtractPrefLenght_StringExtracted();
//FbExtrctAnyStringTests_ExtractPrefLenghtToLong_EmptyString();

METHOD INTERNAL FbExtrctAnyStringTests_ExtractPrefLenght_StringExtracted 
VAR_INST
	fbSut 	: FB_ExtractAnyString;
	sDataString		: T_LongSTRING := 'ABCDEFGHIJKL'; 
	sResult : T_LongSTRING;	// Result
END_VAR
//FB_ExtractAnyString
TEST('FbExtrctAnyStringTests_ExtractPrefLenght_StringExtracted');

fbSut(
	bExtractData:= TRUE, 
	nExtractChars:= 3 , 
	sPrefix:='E' , 
	sSuffix:= '', 
	bIgnoreCase:= FALSE, 
	eExtractMode := E_STRING_ExtrMode.WITHOUTIDENT_PURGE, 
	sDataString:= sDataString, 
	bStringFound=> , 
	sExtractedString=>sResult, 
	nExtractedStringPos=> ,
	nExtractedStringLen=> ,
	nDataStringLen=> );
	
	
	AssertEquals_STRING(	Expected:= 'FGH', 
						Actual:= fbSut.sExtractedString, 
						Message:= 'Extracted string is not as expected');
						
	AssertEquals_STRING(	Expected:= 'IJKL', 
						Actual:= sDataString, 
						Message:= 'Remaining string is not as expected');
						
TEST_FINISHED();
END_METHOD

METHOD INTERNAL FbExtrctAnyStringTests_ExtractPrefLenghtToLong_EmptyString 
VAR_INST
	fbSut 	: FB_ExtractAnyString;
	sDataString		: T_LongSTRING := 'ABCDEFGHIJKL'; 
	sResult : T_LongSTRING;	// Result
END_VAR
//FB_ExtractAnyString
TEST('FbExtrctAnyStringTests_ExtractPrefLenghtToLong_EmptyString');

fbSut(
	bExtractData:= TRUE, 
	nExtractChars:= 15 , 
	sPrefix:='B' , 
	sSuffix:= '', 
	bIgnoreCase:= FALSE, 
	eExtractMode := E_STRING_ExtrMode.WITHOUTIDENT_PURGE, 
	sDataString:= sDataString, 
	bStringFound=> , 
	sExtractedString=>sResult, 
	nExtractedStringPos=> ,
	nExtractedStringLen=> ,
	nDataStringLen=> );
	
	
	AssertEquals_STRING(	Expected:= 'CDEFGHIJKL', 
						Actual:= fbSut.sExtractedString, 
						Message:= 'Extracted string is not as expected');
						
	AssertEquals_STRING(	Expected:= '', 
						Actual:= sDataString, 
						Message:= 'Remaining string is not as expected');
						
TEST_FINISHED();
END_METHOD

METHOD INTERNAL testMain01_ModeWITHIDENT_ExactDataNoPurge
VAR
	fbSut 			: FB_ExtractAnyString;
	sDataString		: T_LongSTRING := '$01ST=53;$02CT=10;DS=]d201062533414058582101485MV125000156300$1D24010120957;OG=3;XP=94;YP=-39;AP=-88;CS=06.2;SC=0070;PN=1;QS=3;$03$04'; 
	sResult 		: T_LongSTRING;	// Result
END_VAR
TEST('testMain01_ModeWITHIDENT_ExactDataNoPurge');

fbSut(
	bExtractData:= TRUE, 
	nExtractChars:=0 , 
	sPrefix:='DS=' , 
	sSuffix:= ';OG', 
	bIgnoreCase:= FALSE, 
	eExtractMode := E_STRING_ExtrMode.WITHIDENT, 
	sDataString:= sDataString, 
	bStringFound=> , 
	sExtractedString=>sResult, 
	nExtractedStringPos=> ,
	nExtractedStringLen=> ,
	nDataStringLen=> );
	
	
	AssertEquals_STRING(	Expected:= 'DS=]d201062533414058582101485MV125000156300$1D24010120957;OG', 
						Actual:= sResult, 
						Message:= 'Extracted string is not as expected');
						
	AssertEquals_STRING(	Expected:= '$01ST=53;$02CT=10;=3;XP=94;YP=-39;AP=-88;CS=06.2;SC=0070;PN=1;QS=3;$03$04', 
						Actual:= sDataString, 
						Message:= 'Remaining string is not as expected');
						
TEST_FINISHED();
END_METHOD

METHOD INTERNAL testMain02_ModeWITHIDENTPURGE_ExactDataAndPurge
VAR
	fbSut 			: FB_ExtractAnyString;
	sDataString		: T_LongSTRING := '$01ST=53;$02CT=10;DS=]d201062533414058582101485MV125000156300$1D24010120957;OG=3;XP=94;YP=-39;AP=-88;CS=06.2;SC=0070;PN=1;QS=3;$03$04'; 
	sResult 		: T_LongSTRING;	// Result
END_VAR
TEST('testMain02_ModeWITHIDENTPURGE_ExactDataAndPurge');

fbSut(
	bExtractData:= TRUE, 
	nExtractChars:=0 , 
	sPrefix:='DS=' , 
	sSuffix:= ';OG', 
	bIgnoreCase:= FALSE, 
	eExtractMode := E_STRING_ExtrMode.WITHIDENT_PURGE, 
	sDataString:= sDataString, 
	bStringFound=> , 
	sExtractedString=>sResult, 
	nExtractedStringPos=> ,
	nExtractedStringLen=> ,
	nDataStringLen=> );
	
	
	AssertEquals_STRING(	Expected:= 'DS=]d201062533414058582101485MV125000156300$1D24010120957;OG', 
						Actual:= sResult, 
						Message:= 'Extracted string is not as expected');
						
	AssertEquals_STRING(	Expected:= '=3;XP=94;YP=-39;AP=-88;CS=06.2;SC=0070;PN=1;QS=3;$03$04', 
						Actual:= sDataString, 
						Message:= 'Remaining string is not as expected');
						
TEST_FINISHED();
END_METHOD

METHOD INTERNAL testMain03_ModeWITHOUTIDENT_ExtractDataNoPurge
VAR
	fbSut 			: FB_ExtractAnyString;
	sDataString		: T_LongSTRING := '$01ST=53;$02CT=10;DS=]d201062533414058582101485MV125000156300$1D24010120957;OG=3;XP=94;YP=-39;AP=-88;CS=06.2;SC=0070;PN=1;QS=3;$03$04'; 
	sResult 		: T_LongSTRING;	// Result
END_VAR
TEST('testMain03_ModeWITHOUTIDENT_ExtractDataNoPurge');

fbSut(
	bExtractData:= TRUE, 
	nExtractChars:=0 , 
	sPrefix:='DS=' , 
	sSuffix:= ';OG', 
	bIgnoreCase:= FALSE, 
	eExtractMode := E_STRING_ExtrMode.WITHOUTIDENT, 
	sDataString:= sDataString, 
	bStringFound=> , 
	sExtractedString=>sResult, 
	nExtractedStringPos=> ,
	nExtractedStringLen=> ,
	nDataStringLen=> );
	
	
	AssertEquals_STRING(	Expected:= ']d201062533414058582101485MV125000156300$1D24010120957', 
						Actual:= sResult, 
						Message:= 'Extracted string is not as expected');
						
	AssertEquals_STRING(	Expected:= '$01ST=53;$02CT=10;DS=;OG=3;XP=94;YP=-39;AP=-88;CS=06.2;SC=0070;PN=1;QS=3;$03$04', 
						Actual:= sDataString, 
						Message:= 'Remaining string is not as expected');
						
TEST_FINISHED();
END_METHOD

METHOD INTERNAL testMain04_ModeWITHOUTIDENTPURGE_ExtractDataAndPurge
VAR
	fbSut 			: FB_ExtractAnyString;
	sDataString		: T_LongSTRING := '$01ST=53;$02CT=10;DS=]d201062533414058582101485MV125000156300$1D24010120957;OG=3;XP=94;YP=-39;AP=-88;CS=06.2;SC=0070;PN=1;QS=3;$03$04'; 
	sResult 		: T_LongSTRING;	// Result
END_VAR
TEST('testMain04_ModeWITHOUTIDENTPURGE_ExtractDataAndPurge');

fbSut(
	bExtractData:= TRUE, 
	nExtractChars:=0 , 
	sPrefix:='DS=' , 
	sSuffix:= ';OG', 
	bIgnoreCase:= FALSE, 
	eExtractMode := E_STRING_ExtrMode.WITHOUTIDENT_PURGE, 
	sDataString:= sDataString, 
	bStringFound=> , 
	sExtractedString=>sResult, 
	nExtractedStringPos=> ,
	nExtractedStringLen=> ,
	nDataStringLen=> );
	
	
	AssertEquals_STRING(	Expected:= ']d201062533414058582101485MV125000156300$1D24010120957', 
						Actual:= sResult, 
						Message:= 'Extracted string is not as expected');
						
	AssertEquals_STRING(	Expected:= ';OG=3;XP=94;YP=-39;AP=-88;CS=06.2;SC=0070;PN=1;QS=3;$03$04', 
						Actual:= sDataString, 
						Message:= 'Remaining string is not as expected');
						
TEST_FINISHED();
END_METHOD

METHOD INTERNAL testMain05_ModeWITHOUTIDENTREMIDENT_ExtractDataNoPurge
VAR
	fbSut 			: FB_ExtractAnyString;
	sDataString		: T_LongSTRING := '$01ST=53;$02CT=10;DS=]d201062533414058582101485MV125000156300$1D24010120957;OG=3;XP=94;YP=-39;AP=-88;CS=06.2;SC=0070;PN=1;QS=3;$03$04'; 
	sResult 		: T_LongSTRING;	// Result
END_VAR
TEST('testMain05_ModeWITHOUTIDENTREMIDENT_ExtractDataNoPurge');

fbSut(
	bExtractData:= TRUE, 
	nExtractChars:=0 , 
	sPrefix:='DS=' , 
	sSuffix:= ';OG', 
	bIgnoreCase:= FALSE, 
	eExtractMode := E_STRING_ExtrMode.WITHOUTIDENT_REMIDENT, 
	sDataString:= sDataString, 
	bStringFound=> , 
	sExtractedString=>sResult, 
	nExtractedStringPos=> ,
	nExtractedStringLen=> ,
	nDataStringLen=> );
	
	
	AssertEquals_STRING(	Expected:= ']d201062533414058582101485MV125000156300$1D24010120957', 
						Actual:= sResult, 
						Message:= 'Extracted string is not as expected');
						
	AssertEquals_STRING(	Expected:= '$01ST=53;$02CT=10;=3;XP=94;YP=-39;AP=-88;CS=06.2;SC=0070;PN=1;QS=3;$03$04', 
						Actual:= sDataString, 
						Message:= 'Remaining string is not as expected');
						
TEST_FINISHED();
END_METHOD

METHOD INTERNAL testMain06_ModeWITHOUTIDENTREMIDENTPURGE_ExtractDataAndPurge
VAR
	fbSut 			: FB_ExtractAnyString;
	sDataString		: T_LongSTRING := '$01ST=53;$02CT=10;DS=]d201062533414058582101485MV125000156300$1D24010120957;OG=3;XP=94;YP=-39;AP=-88;CS=06.2;SC=0070;PN=1;QS=3;$03$04'; 
	sResult 		: T_LongSTRING;	// Result
END_VAR
TEST('testMain06_ModeWITHOUTIDENTREMIDENTPURGE_ExtractDataAndPurge');

fbSut(
	bExtractData:= TRUE, 
	nExtractChars:=0 , 
	sPrefix:='DS=' , 
	sSuffix:= ';OG', 
	bIgnoreCase:= FALSE, 
	eExtractMode := E_STRING_ExtrMode.WITHOUTIDENT_REMIDENT_PURGE, 
	sDataString:= sDataString, 
	bStringFound=> , 
	sExtractedString=>sResult, 
	nExtractedStringPos=> ,
	nExtractedStringLen=> ,
	nDataStringLen=> );
	
	
	AssertEquals_STRING(	Expected:= ']d201062533414058582101485MV125000156300$1D24010120957', 
						Actual:= sResult, 
						Message:= 'Extracted string is not as expected');
						
	AssertEquals_STRING(	Expected:= '=3;XP=94;YP=-39;AP=-88;CS=06.2;SC=0070;PN=1;QS=3;$03$04', 
						Actual:= sDataString, 
						Message:= 'Remaining string is not as expected');
						
TEST_FINISHED();
END_METHOD

METHOD INTERNAL testMain07_ExtractFromLongString_ExtractData
VAR
	fbSut 			: FB_ExtractAnyString;
	sResult 		: T_LongSTRING;	// Result
END_VAR
VAR_INST
	aDataString		: ARRAY[1..3] OF T_LongSTRING;
END_VAR

// '$01ST=53;$02CT=10;DS=GZDNP5JOA3IL;OG=3;XP=-50;YP=50;AP=-88;CS=06.2;SC=0070;QS=3;PN=1;$03$04
//		$01ST=53;$02CT=10;DS=N7E1Y89UNK3O;OG=3;XP=-50;YP=-50;AP=-88;CS=06.2;SC=0070;QS=3;PN=2;$03$04
//		$01ST=53;$02CT=10;DS=JHWJXYFNX9DS;OG=3;XP=50;YP=50;AP=-88;CS=06.2;SC=0070;QS=3;PN=3;$03$04
//		$01ST=53;$02CT=10;DS=XGBEZLBV8A9I;OG=3;XP=50;YP=-50;AP=-88;CS=06.2;SC=0070;QS=3;PN=4;$03$04';
TEST('testMain07_ExtractFromLongString_ExtractData');	
			
aDataString[1] := '$01ST=53;$02CT=10;DS=GZDNP5JOA3IL;OG=3;XP=-50;YP=50;AP=-88;CS=06.2;SC=0070;QS=3;PN=1;$03$04
					$01ST=53;$02CT=10;DS=N7E1Y89UNK3O;OG=3;XP=-50;YP=-50;AP=-88;CS=06.2;SC=0070;QS=3;PN=2;$03$04
					$01ST=53;$02CT=10;DS=JHWJXYFNX9DS;OG=3;XP=50;YP=50;AP=-88;CS=06.2;SC=0070;QS=3;PN=3;$03$04
					$01ST=53;$02CT=10;DS=XGBEZLBV8A9I;OG=3;XP=50;YP=-50;AP=-88;CS=06.2;SC=0070;QS=3;PN=4;$03$04'; 
fbSut(
	bExtractData:= TRUE, 
	nExtractChars:=9 , 
	sPrefix:='XGB' , 
	sSuffix:= '', 
	bIgnoreCase:= FALSE, 
	eExtractMode := E_STRING_ExtrMode.WITHIDENT, 
	sDataString:= aDataString[1], 
	bStringFound=> , 
	sExtractedString=>sResult, 
	nExtractedStringPos=> ,
	nExtractedStringLen=> ,
	nDataStringLen=> );
	
	
	AssertEquals_STRING(	Expected:= 'XGBEZLBV8A9I', 
						Actual:= sResult, 
						Message:= 'Extr data in mode:WITHIDENT not as expect');
	
aDataString[2] := '$01ST=53;$02CT=10;DS=GZDNP5JOA3IL;OG=3;XP=-50;YP=50;AP=-88;CS=06.2;SC=0070;QS=3;PN=1;$03$04
					$01ST=53;$02CT=10;DS=N7E1Y89UNK3O;OG=3;XP=-50;YP=-50;AP=-88;CS=06.2;SC=0070;QS=3;PN=2;$03$04
					$01ST=53;$02CT=10;DS=JHWJXYFNX9DS;OG=3;XP=50;YP=50;AP=-88;CS=06.2;SC=0070;QS=3;PN=3;$03$04
					$01ST=53;$02CT=10;DS=XGBEZLBV8A9I;OG=3;XP=50;YP=-50;AP=-88;CS=06.2;SC=0070;QS=3;PN=4;$03$04'; 
					
fbSut(
	bExtractData:= TRUE, 
	nExtractChars:=0 , 
	sPrefix:='DS=' , 
	sSuffix:= ';OG', 
	bIgnoreCase:= FALSE, 
	eExtractMode := E_STRING_ExtrMode.WITHOUTIDENT_PURGE, 
	sDataString:= aDataString[2], 
	bStringFound=> , 
	sExtractedString=>sResult, 
	nExtractedStringPos=> ,
	nExtractedStringLen=> ,
	nDataStringLen=> );
	
	
	AssertEquals_STRING(	Expected:= 'GZDNP5JOA3IL', 
						Actual:= sResult, 
						Message:= 'Extr data in mode:WITHOUTIDENT_PURGE not as expect');
				
TEST_FINISHED();
END_METHOD

METHOD INTERNAL testMain08_ExtractFromLongString_LenghtExtractedDataOk
VAR
	fbSut 			: FB_ExtractAnyString;
	nResult 		: UDINT;	// Result
END_VAR
VAR_INST
	aDataString		: ARRAY[1..4] OF T_LongSTRING;
END_VAR
TEST('testMain08_ExtractFromLongString_LenghtExtractedDataOk');	
			
aDataString[1] := '$01ST=53;$02CT=10;DS=GZDNP5JOA3IL;OG=3;XP=-50;YP=50;AP=-88;CS=06.2;SC=0070;QS=3;PN=1;$03$04
					$01ST=53;$02CT=10;DS=N7E1Y89UNK3O;OG=3;XP=-50;YP=-50;AP=-88;CS=06.2;SC=0070;QS=3;PN=2;$03$04
					$01ST=53;$02CT=10;DS=JHWJXYFNX9DS;OG=3;XP=50;YP=50;AP=-88;CS=06.2;SC=0070;QS=3;PN=3;$03$04
					$01ST=53;$02CT=10;DS=XGBEZLBV8A9I;OG=3;XP=50;YP=-50;AP=-88;CS=06.2;SC=0070;QS=3;PN=4;$03$04'; 
					
